LIN {X 0,Y 445.877,Z 691.903,A -85,B 0,C 180,E1 -8721.844,E2 -8721.844} C_VEL
LIN {X 0,Y 445.652,Z 697.529,A -85,B 0,C 180,E1 -8723.208,E2 -8723.208} C_VEL
LIN {X 0,Y 445.575,Z 701.931,A -85,B 0,C 180,E1 -8724.569,E2 -8724.569} C_VEL
LIN {X 0,Y 445.476,Z 704.248,A -85,B 0,C 180,E1 -8725.476,E2 -8725.476} C_VEL
LIN {X 0,Y 445.468,Z 706.135,A -85,B 0,C 180,E1 -8726.382,E2 -8726.382} C_VEL
LIN {X 0,Y 445.487,Z 707.56,A -85,B 0,C 180,E1 -8727.287,E2 -8727.287} C_VEL
LIN {X 0,Y 445.395,Z 709.177,A -85,B 0,C 180,E1 -8729.096,E2 -8729.096} C_VEL
LIN {X 0,Y 445.415,Z 709.398,A -85,B 0,C 180,E1 -8730,E2 -8730} C_VEL
LIN {X 0,Y 445.434,Z 709.177,A -85,B 0,C 180,E1 -8730.904,E2 -8730.904} C_VEL
LIN {X 0,Y 445.493,Z 707.56,A -85,B 0,C 180,E1 -8732.713,E2 -8732.713} C_VEL
LIN {X 0,Y 445.478,Z 706.134,A -85,B 0,C 180,E1 -8733.618,E2 -8733.618} C_VEL
LIN {X 0,Y 445.558,Z 703.166,A -85,B 0,C 180,E1 -8734.977,E2 -8734.977} C_VEL
LIN {X 0,Y 445.627,Z 698.572,A -85,B 0,C 180,E1 -8736.496,E2 -8736.496} C_VEL
LIN {X 0,Y 445.881,Z 691.901,A -85,B 0,C 180,E1 -8738.155,E2 -8738.155} C_VEL
LIN {X 0,Y 446.193,Z 684.816,A -85,B 0,C 180,E1 -8739.52,E2 -8739.52} C_VEL
LIN {X 0,Y 446.626,Z 675.955,A -85,B 0,C 180,E1 -8740.884,E2 -8740.884} C_VEL
LIN {X 0,Y 447.161,Z 666.837,A -85,B 0,C 180,E1 -8742.02,E2 -8742.02} C_VEL
LIN {X 0,Y 447.743,Z 655.911,A -85,B 0,C 180,E1 -8743.108,E2 -8743.108} C_VEL
LIN {X 0,Y 448.243,Z 645.348,A -85,B 0,C 180,E1 -8743.949,E2 -8743.949} C_VEL
LIN {X 0,Y 448.735,Z 633.519,A -85,B 0,C 180,E1 -8744.686,E2 -8744.686} C_VEL
LIN {X 0,Y 449.209,Z 620.349,A -85,B 0,C 180,E1 -8745.279,E2 -8745.279} C_VEL
LIN {X 0,Y 449.541,Z 608.315,A -85,B 0,C 180,E1 -8745.645,E2 -8745.645} C_VEL
LIN {X 0,Y 449.98,Z 567.208,A -85,B 0,C 180,E1 -8746.328,E2 -8746.328} C_VEL
LIN {X 0,Y 450.253,Z 534.372,A -85,B 0,C 180,E1 -8746.887,E2 -8746.887} C_VEL
LIN {X 0,Y 450.479,Z 513.135,A -85,B 0,C 180,E1 -8747.309,E2 -8747.309} C_VEL
LIN {X 0,Y 447.627,Z 483.502,A -85,B 0,C 180,E1 -8748.061,E2 -8748.061} C_VEL
LIN {X 0,Y 447.327,Z 480.598,A -85,B 0,C 180,E1 -8748.184,E2 -8748.184} C_VEL
LIN {X 0,Y 448.232,Z 456.008,A -85,B 0,C 180,E1 -8751.621,E2 -8751.621} C_VEL
LIN {X 0,Y 449.365,Z 434.276,A -85,B 0,C 180,E1 -8754.758,E2 -8754.758} C_VEL
LIN {X 0,Y 450.768,Z 413.421,A -85,B 0,C 180,E1 -8757.887,E2 -8757.887} C_VEL
LIN {X 0,Y 449.482,Z 405.511,A -85,B 0,C 180,E1 -8759.25,E2 -8759.25} C_VEL
LIN {X 0,Y 446.902,Z 394.819,A -85,B 0,C 180,E1 -8761.263,E2 -8761.263} C_VEL
LIN {X 0,Y 446.417,Z 392.958,A -85,B 0,C 180,E1 -8761.686,E2 -8761.686} C_VEL
LIN {X 0,Y 446.412,Z 392.881,A -85,B 0,C 180,E1 -8764.525,E2 -8764.525} C_VEL
LIN {X 0,Y 446.389,Z 392.884,A -85,B 0,C 180,E1 -8767.881,E2 -8767.881} C_VEL
LIN {X 0,Y 446.395,Z 392.878,A -85,B 0,C 180,E1 -8770.913,E2 -8770.913} C_VEL
LIN {X 0,Y 446.391,Z 392.882,A -85,B 0,C 180,E1 -8773.847,E2 -8773.847} C_VEL
LIN {X 0,Y 446.386,Z 392.879,A -85,B 0,C 180,E1 -8776.405,E2 -8776.405} C_VEL
LIN {X 0,Y 446.399,Z 392.88,A -85,B 0,C 180,E1 -8779.797,E2 -8779.797} C_VEL
LIN {X 0,Y 446.396,Z 392.882,A -85,B 0,C 180,E1 -8783.254,E2 -8783.254} C_VEL
LIN {X 0,Y 446.45,Z 392.872,A -85,B 0,C 180,E1 -8786.566,E2 -8786.566} C_VEL
LIN {X 0,Y 446.43,Z 392.877,A -85,B 0,C 180,E1 -8789.98,E2 -8789.98} C_VEL
LIN {X 0,Y 446.447,Z 392.873,A -85,B 0,C 180,E1 -8792.837,E2 -8792.837} C_VEL
LIN {X 0,Y 446.463,Z 392.873,A -85,B 0,C 180,E1 -8795.925,E2 -8795.925} C_VEL
LIN {X 0,Y 446.456,Z 392.874,A -85,B 0,C 180,E1 -8798.773,E2 -8798.773} C_VEL
LIN {X 0,Y 446.504,Z 392.971,A -85,B 0,C 180,E1 -8802.173,E2 -8802.173} C_VEL
LIN {X 0,Y 446.675,Z 393.84,A -85,B 0,C 180,E1 -8802.346,E2 -8802.346} C_VEL
LIN {X 0,Y 451.59,Z 405.892,A -85,B 0,C 180,E1 -8802.9,E2 -8802.9} C_VEL
LIN {X 0,Y 450.382,Z 476.779,A -85,B 0,C 180,E1 -8804.327,E2 -8804.327} C_VEL
LIN {X 0,Y 450.3,Z 489.562,A -85,B 0,C 180,E1 -8804.73,E2 -8804.73} C_VEL
LIN {X 0,Y 450.103,Z 503.008,A -85,B 0,C 180,E1 -8805.359,E2 -8805.359} C_VEL
LIN {X 0,Y 449.851,Z 513.751,A -85,B 0,C 180,E1 -8806.03,E2 -8806.03} C_VEL
LIN {X 0,Y 449.45,Z 524.679,A -85,B 0,C 180,E1 -8806.895,E2 -8806.895} C_VEL
LIN {X 0,Y 448.972,Z 533.964,A -85,B 0,C 180,E1 -8807.8,E2 -8807.8} C_VEL
LIN {X 0,Y 448.559,Z 543.404,A -85,B 0,C 180,E1 -8808.934,E2 -8808.934} C_VEL
LIN {X 0,Y 448.065,Z 551.12,A -85,B 0,C 180,E1 -8810.065,E2 -8810.065} C_VEL
LIN {X 0,Y 447.706,Z 558.821,A -85,B 0,C 180,E1 -8811.48,E2 -8811.48} C_VEL
LIN {X 0,Y 447.329,Z 564.472,A -85,B 0,C 180,E1 -8812.78,E2 -8812.78} C_VEL
LIN {X 0,Y 447.07,Z 569.094,A -85,B 0,C 180,E1 -8814.135,E2 -8814.135} C_VEL
LIN {X 0,Y 446.694,Z 572.607,A -85,B 0,C 180,E1 -8815.488,E2 -8815.488} C_VEL
LIN {X 0,Y 446.742,Z 574.35,A -85,B 0,C 180,E1 -8816.392,E2 -8816.392} C_VEL
LIN {X 0,Y 446.596,Z 575.652,A -85,B 0,C 180,E1 -8817.294,E2 -8817.294} C_VEL
LIN {X 0,Y 446.502,Z 576.521,A -85,B 0,C 180,E1 -8818.196,E2 -8818.196} C_VEL
LIN {X 0,Y 446.405,Z 576.994,A -85,B 0,C 180,E1 -8819.098,E2 -8819.098} C_VEL
LIN {X 0,Y 446.363,Z 577.045,A -85,B 0,C 180,E1 -8820,E2 -8820} C_VEL
LIN {X 0,Y 446.38,Z 576.645,A -85,B 0,C 180,E1 -8820.902,E2 -8820.902} C_VEL
LIN {X 0,Y 446.301,Z 575.861,A -85,B 0,C 180,E1 -8821.805,E2 -8821.805} C_VEL
LIN {X 0,Y 446.424,Z 574.653,A -85,B 0,C 180,E1 -8822.707,E2 -8822.707} C_VEL
LIN {X 0,Y 446.411,Z 572.035,A -85,B 0,C 180,E1 -8824.063,E2 -8824.063} C_VEL
LIN {X 0,Y 446.568,Z 568.375,A -85,B 0,C 180,E1 -8825.418,E2 -8825.418} C_VEL
LIN {X 0,Y 446.892,Z 562.968,A -85,B 0,C 180,E1 -8826.919,E2 -8826.919} C_VEL
LIN {X 0,Y 447.153,Z 556.334,A -85,B 0,C 180,E1 -8828.36,E2 -8828.36} C_VEL
LIN {X 0,Y 447.458,Z 548.495,A -85,B 0,C 180,E1 -8829.721,E2 -8829.721} C_VEL
LIN {X 0,Y 447.788,Z 540.446,A -85,B 0,C 180,E1 -8830.856,E2 -8830.856} C_VEL
LIN {X 0,Y 448.184,Z 530.608,A -85,B 0,C 180,E1 -8831.992,E2 -8831.992} C_VEL
LIN {X 0,Y 448.612,Z 519.67,A -85,B 0,C 180,E1 -8833.015,E2 -8833.015} C_VEL
LIN {X 0,Y 448.905,Z 508.7,A -85,B 0,C 180,E1 -8833.836,E2 -8833.836} C_VEL
LIN {X 0,Y 449.181,Z 496.311,A -85,B 0,C 180,E1 -8834.556,E2 -8834.556} C_VEL
LIN {X 0,Y 449.417,Z 483.722,A -85,B 0,C 180,E1 -8835.098,E2 -8835.098} C_VEL
LIN {X 0,Y 449.495,Z 470.727,A -85,B 0,C 180,E1 -8835.473,E2 -8835.473} C_VEL
LIN {X 0,Y 450.128,Z 404.106,A -85,B 0,C 180,E1 -8836.708,E2 -8836.708} C_VEL
LIN {X 0,Y 446.657,Z 393.7,A -85,B 0,C 180,E1 -8837.05,E2 -8837.05} C_VEL
LIN {X 0,Y 446.482,Z 392.961,A -85,B 0,C 180,E1 -8837.209,E2 -8837.209} C_VEL
LIN {X 0,Y 446.447,Z 392.875,A -85,B 0,C 180,E1 -8840.263,E2 -8840.263} C_VEL
LIN {X 0,Y 446.431,Z 392.876,A -85,B 0,C 180,E1 -8843.177,E2 -8843.177} C_VEL
LIN {X 0,Y 446.441,Z 392.873,A -85,B 0,C 180,E1 -8846.193,E2 -8846.193} C_VEL
LIN {X 0,Y 446.44,Z 392.868,A -85,B 0,C 180,E1 -8849.21,E2 -8849.21} C_VEL
LIN {X 0,Y 446.422,Z 392.877,A -85,B 0,C 180,E1 -8852.362,E2 -8852.362} C_VEL
LIN {X 0,Y 446.42,Z 392.874,A -85,B 0,C 180,E1 -8855.626,E2 -8855.626} C_VEL
LIN {X 0,Y 446.443,Z 392.874,A -85,B 0,C 180,E1 -8859.027,E2 -8859.027} C_VEL
LIN {X 0,Y 446.423,Z 392.872,A -85,B 0,C 180,E1 -8862.275,E2 -8862.275} C_VEL
LIN {X 0,Y 446.452,Z 392.869,A -85,B 0,C 180,E1 -8865.104,E2 -8865.104} C_VEL
LIN {X 0,Y 446.421,Z 392.877,A -85,B 0,C 180,E1 -8868.608,E2 -8868.608} C_VEL
LIN {X 0,Y 446.413,Z 392.865,A -85,B 0,C 180,E1 -8871.922,E2 -8871.922} C_VEL
LIN {X 0,Y 446.431,Z 392.869,A -85,B 0,C 180,E1 -8875.477,E2 -8875.477} C_VEL
LIN {X 0,Y 446.488,Z 392.994,A -85,B 0,C 180,E1 -8879.117,E2 -8879.117} C_VEL
LIN {X 0,Y 449.858,Z 407.067,A -85,B 0,C 180,E1 -8881.314,E2 -8881.314} C_VEL
LIN {X 0,Y 451.299,Z 414.583,A -85,B 0,C 180,E1 -8882.448,E2 -8882.448} C_VEL
LIN {X 0,Y 450.315,Z 437.381,A -85,B 0,C 180,E1 -8885.57,E2 -8885.57} C_VEL
LIN {X 0,Y 449.475,Z 456.758,A -85,B 0,C 180,E1 -8888.201,E2 -8888.201} C_VEL
LIN {X 0,Y 448.796,Z 474.172,A -85,B 0,C 180,E1 -8890.501,E2 -8890.501} C_VEL
LIN {X 0,Y 448.016,Z 477.382,A -85,B 0,C 180,E1 -8890.88,E2 -8890.88} C_VEL
LIN {X 0,Y 444.945,Z 482.695,A -85,B 0,C 180,E1 -8891.434,E2 -8891.434} C_VEL
LIN {X 0,Y 442.344,Z 487.283,A -85,B 0,C 180,E1 -8891.854,E2 -8891.854} C_VEL
LIN {X 0,Y 441.926,Z 490.019,A -85,B 0,C 180,E1 -8891.993,E2 -8891.993} C_VEL
LIN {X 0,Y 441.979,Z 490.598,A -85,B 0,C 180,E1 -8892.008,E2 -8892.008} C_VEL
LIN {X 0,Y 444.18,Z 506.961,A -85,B 0,C 180,E1 -8892.374,E2 -8892.374} C_VEL
LIN {X 0,Y 443.246,Z 598.809,A -85,B 0,C 180,E1 -8893.89,E2 -8893.89} C_VEL
LIN {X 0,Y 442.885,Z 612.281,A -85,B 0,C 180,E1 -8894.291,E2 -8894.291} C_VEL
LIN {X 0,Y 442.359,Z 624.85,A -85,B 0,C 180,E1 -8894.862,E2 -8894.862} C_VEL
LIN {X 0,Y 441.775,Z 636.976,A -85,B 0,C 180,E1 -8895.607,E2 -8895.607} C_VEL
LIN {X 0,Y 441.233,Z 648.191,A -85,B 0,C 180,E1 -8896.504,E2 -8896.504} C_VEL
LIN {X 0,Y 440.634,Z 658.741,A -85,B 0,C 180,E1 -8897.566,E2 -8897.566} C_VEL
LIN {X 0,Y 439.971,Z 668.052,A -85,B 0,C 180,E1 -8898.716,E2 -8898.716} C_VEL
LIN {X 0,Y 439.426,Z 677.035,A -85,B 0,C 180,E1 -8900.1,E2 -8900.1} C_VEL
LIN {X 0,Y 438.986,Z 684.246,A -85,B 0,C 180,E1 -8901.484,E2 -8901.484} C_VEL
LIN {X 0,Y 438.719,Z 689.142,A -85,B 0,C 180,E1 -8902.637,E2 -8902.637} C_VEL
LIN {X 0,Y 438.555,Z 693.879,A -85,B 0,C 180,E1 -8904.021,E2 -8904.021} C_VEL
LIN {X 0,Y 438.375,Z 697.508,A -85,B 0,C 180,E1 -8905.402,E2 -8905.402} C_VEL
LIN {X 0,Y 438.307,Z 699.376,A -85,B 0,C 180,E1 -8906.323,E2 -8906.323} C_VEL
LIN {X 0,Y 438.346,Z 700.805,A -85,B 0,C 180,E1 -8907.243,E2 -8907.243} C_VEL
LIN {X 0,Y 438.231,Z 702.424,A -85,B 0,C 180,E1 -8909.081,E2 -8909.081} C_VEL
LIN {X 0,Y 438.229,Z 702.662,A -85,B 0,C 180,E1 -8910,E2 -8910} C_VEL
LIN {X 0,Y 438.231,Z 702.471,A -85,B 0,C 180,E1 -8910.919,E2 -8910.919} C_VEL
LIN {X 0,Y 438.346,Z 700.914,A -85,B 0,C 180,E1 -8912.757,E2 -8912.757} C_VEL
LIN {X 0,Y 438.307,Z 699.546,A -85,B 0,C 180,E1 -8913.677,E2 -8913.677} C_VEL
LIN {X 0,Y 438.448,Z 696.666,A -85,B 0,C 180,E1 -8915.058,E2 -8915.058} C_VEL
LIN {X 0,Y 438.547,Z 692.602,A -85,B 0,C 180,E1 -8916.488,E2 -8916.488} C_VEL
LIN {X 0,Y 438.766,Z 687.691,A -85,B 0,C 180,E1 -8917.825,E2 -8917.825} C_VEL
LIN {X 0,Y 439.161,Z 681.306,A -85,B 0,C 180,E1 -8919.209,E2 -8919.209} C_VEL
LIN {X 0,Y 439.625,Z 673.378,A -85,B 0,C 180,E1 -8920.594,E2 -8920.594} C_VEL
LIN {X 0,Y 440.164,Z 665.28,A -85,B 0,C 180,E1 -8921.746,E2 -8921.746} C_VEL
LIN {X 0,Y 440.869,Z 655.338,A -85,B 0,C 180,E1 -8922.896,E2 -8922.896} C_VEL
LIN {X 0,Y 441.388,Z 644.17,A -85,B 0,C 180,E1 -8923.936,E2 -8923.936} C_VEL
LIN {X 0,Y 441.985,Z 633.248,A -85,B 0,C 180,E1 -8924.739,E2 -8924.739} C_VEL
LIN {X 0,Y 442.566,Z 620.993,A -85,B 0,C 180,E1 -8925.426,E2 -8925.426} C_VEL
LIN {X 0,Y 443.06,Z 608.283,A -85,B 0,C 180,E1 -8925.939,E2 -8925.939} C_VEL
LIN {X 0,Y 443.367,Z 594.914,A -85,B 0,C 180,E1 -8926.283,E2 -8926.283} C_VEL
LIN {X 0,Y 444.09,Z 505.201,A -85,B 0,C 180,E1 -8927.753,E2 -8927.753} C_VEL
LIN {X 0,Y 441.619,Z 487.767,A -85,B 0,C 180,E1 -8928.168,E2 -8928.168} C_VEL
LIN {X 0,Y 442.206,Z 467.995,A -85,B 0,C 180,E1 -8930.709,E2 -8930.709} C_VEL
LIN {X 0,Y 443.215,Z 444.829,A -85,B 0,C 180,E1 -8933.851,E2 -8933.851} C_VEL
LIN {X 0,Y 444.211,Z 423.493,A -85,B 0,C 180,E1 -8936.802,E2 -8936.802} C_VEL
LIN {X 0,Y 444.469,Z 415.37,A -85,B 0,C 180,E1 -8937.929,E2 -8937.929} C_VEL
LIN {X 0,Y 441.016,Z 400.06,A -85,B 0,C 180,E1 -8940.285,E2 -8940.285} C_VEL
LIN {X 0,Y 439.416,Z 393.899,A -85,B 0,C 180,E1 -8941.286,E2 -8941.286} C_VEL
LIN {X 0,Y 439.387,Z 393.749,A -85,B 0,C 180,E1 -8944.044,E2 -8944.044} C_VEL
LIN {X 0,Y 439.341,Z 393.751,A -85,B 0,C 180,E1 -8946.885,E2 -8946.885} C_VEL
LIN {X 0,Y 439.348,Z 393.748,A -85,B 0,C 180,E1 -8949.84,E2 -8949.84} C_VEL
LIN {X 0,Y 439.335,Z 393.758,A -85,B 0,C 180,E1 -8952.62,E2 -8952.62} C_VEL
LIN {X 0,Y 439.379,Z 393.738,A -85,B 0,C 180,E1 -8955.268,E2 -8955.268} C_VEL
LIN {X 0,Y 439.369,Z 393.753,A -85,B 0,C 180,E1 -8958.747,E2 -8958.747} C_VEL
LIN {X 0,Y 439.362,Z 393.757,A -85,B 0,C 180,E1 -8961.611,E2 -8961.611} C_VEL
LIN {X 0,Y 439.397,Z 393.749,A -85,B 0,C 180,E1 -8964.844,E2 -8964.844} C_VEL
LIN {X 0,Y 439.373,Z 393.755,A -85,B 0,C 180,E1 -8968.139,E2 -8968.139} C_VEL
LIN {X 0,Y 439.385,Z 393.746,A -85,B 0,C 180,E1 -8971.324,E2 -8971.324} C_VEL
LIN {X 0,Y 439.374,Z 393.752,A -85,B 0,C 180,E1 -8974.413,E2 -8974.413} C_VEL
LIN {X 0,Y 439.367,Z 393.748,A -85,B 0,C 180,E1 -8977.425,E2 -8977.425} C_VEL
LIN {X 0,Y 439.445,Z 393.74,A -85,B 0,C 180,E1 -8980.663,E2 -8980.663} C_VEL
LIN {X 0,Y 439.424,Z 393.747,A -85,B 0,C 180,E1 -8984.223,E2 -8984.223} C_VEL
LIN {X 0,Y 439.488,Z 393.737,A -85,B 0,C 180,E1 -8987.286,E2 -8987.286} C_VEL
LIN {X 0,Y 439.479,Z 393.736,A -85,B 0,C 180,E1 -8990.798,E2 -8990.798} C_VEL
LIN {X 0,Y 439.562,Z 393.729,A -85,B 0,C 180,E1 -8993.574,E2 -8993.574} C_VEL
LIN {X 0,Y 439.406,Z 393.737,A -85,B 0,C 180,E1 -8995.413,E2 -8995.413} C_VEL
LIN {X 0,Y 439.629,Z 393.722,A -85,B 0,C 180,E1 -8998.168,E2 -8998.168} C_VEL
LIN {X 0,Y 439.672,Z 393.714,A -85,B 0,C 180,E1 -9000,E2 -9000} C_VEL
LIN {X 0,Y 439.607,Z 393.708,A -85,B 0,C 180,E1 -9002.749,E2 -9002.749} C_VEL
LIN {X 0,Y 439.562,Z 393.728,A -85,B 0,C 180,E1 -9006.426,E2 -9006.426} C_VEL
LIN {X 0,Y 439.478,Z 393.731,A -85,B 0,C 180,E1 -9009.202,E2 -9009.202} C_VEL
LIN {X 0,Y 439.467,Z 393.739,A -85,B 0,C 180,E1 -9012.938,E2 -9012.938} C_VEL
LIN {X 0,Y 439.399,Z 393.736,A -85,B 0,C 180,E1 -9016.325,E2 -9016.325} C_VEL
LIN {X 0,Y 439.372,Z 393.755,A -85,B 0,C 180,E1 -9019.628,E2 -9019.628} C_VEL
LIN {X 0,Y 439.362,Z 393.742,A -85,B 0,C 180,E1 -9022.576,E2 -9022.576} C_VEL
LIN {X 0,Y 439.357,Z 393.756,A -85,B 0,C 180,E1 -9025.588,E2 -9025.588} C_VEL
LIN {X 0,Y 439.384,Z 393.74,A -85,B 0,C 180,E1 -9028.676,E2 -9028.676} C_VEL
LIN {X 0,Y 439.368,Z 393.756,A -85,B 0,C 180,E1 -9032.029,E2 -9032.029} C_VEL
LIN {X 0,Y 439.389,Z 393.745,A -85,B 0,C 180,E1 -9035.338,E2 -9035.338} C_VEL
LIN {X 0,Y 439.35,Z 393.749,A -85,B 0,C 180,E1 -9038.599,E2 -9038.599} C_VEL
LIN {X 0,Y 439.346,Z 393.732,A -85,B 0,C 180,E1 -9042.21,E2 -9042.21} C_VEL
LIN {X 0,Y 439.373,Z 393.753,A -85,B 0,C 180,E1 -9045.267,E2 -9045.267} C_VEL
LIN {X 0,Y 439.359,Z 393.729,A -85,B 0,C 180,E1 -9048.748,E2 -9048.748} C_VEL
LIN {X 0,Y 439.353,Z 393.756,A -85,B 0,C 180,E1 -9051.612,E2 -9051.612} C_VEL
LIN {X 0,Y 439.388,Z 393.753,A -85,B 0,C 180,E1 -9054.843,E2 -9054.843} C_VEL
LIN {X 0,Y 439.389,Z 393.934,A -85,B 0,C 180,E1 -9058.359,E2 -9058.359} C_VEL
LIN {X 0,Y 443.711,Z 412.535,A -85,B 0,C 180,E1 -9061.407,E2 -9061.407} C_VEL
LIN {X 0,Y 444.061,Z 417.576,A -85,B 0,C 180,E1 -9062.171,E2 -9062.171} C_VEL
LIN {X 0,Y 442.664,Z 439.939,A -85,B 0,C 180,E1 -9065.383,E2 -9065.383} C_VEL
LIN {X 0,Y 441.484,Z 462.058,A -85,B 0,C 180,E1 -9068.522,E2 -9068.522} C_VEL
LIN {X 0,Y 440.487,Z 486.126,A -85,B 0,C 180,E1 -9071.888,E2 -9071.888} C_VEL
LIN {X 0,Y 440.734,Z 489.285,A -85,B 0,C 180,E1 -9072.018,E2 -9072.018} C_VEL
LIN {X 0,Y 443.561,Z 515.823,A -85,B 0,C 180,E1 -9072.577,E2 -9072.577} C_VEL
LIN {X 0,Y 442.755,Z 607.315,A -85,B 0,C 180,E1 -9074.079,E2 -9074.079} C_VEL
LIN {X 0,Y 442.367,Z 620.411,A -85,B 0,C 180,E1 -9074.478,E2 -9074.478} C_VEL
LIN {X 0,Y 441.883,Z 633.544,A -85,B 0,C 180,E1 -9075.081,E2 -9075.081} C_VEL
LIN {X 0,Y 441.325,Z 645.346,A -85,B 0,C 180,E1 -9075.827,E2 -9075.827} C_VEL
LIN {X 0,Y 440.771,Z 656.588,A -85,B 0,C 180,E1 -9076.743,E2 -9076.743} C_VEL
LIN {X 0,Y 440.167,Z 666.82,A -85,B 0,C 180,E1 -9077.786,E2 -9077.786} C_VEL
LIN {X 0,Y 439.64,Z 675.926,A -85,B 0,C 180,E1 -9078.94,E2 -9078.94} C_VEL
LIN {X 0,Y 439.166,Z 684.77,A -85,B 0,C 180,E1 -9080.326,E2 -9080.326} C_VEL
LIN {X 0,Y 438.841,Z 691.853,A -85,B 0,C 180,E1 -9081.713,E2 -9081.713} C_VEL
LIN {X 0,Y 438.588,Z 697.476,A -85,B 0,C 180,E1 -9083.097,E2 -9083.097} C_VEL
LIN {X 0,Y 438.49,Z 701.879,A -85,B 0,C 180,E1 -9084.481,E2 -9084.481} C_VEL
LIN {X 0,Y 438.403,Z 704.195,A -85,B 0,C 180,E1 -9085.402,E2 -9085.402} C_VEL
LIN {X 0,Y 438.366,Z 706.082,A -85,B 0,C 180,E1 -9086.323,E2 -9086.323} C_VEL
LIN {X 0,Y 438.412,Z 707.507,A -85,B 0,C 180,E1 -9087.243,E2 -9087.243} C_VEL
LIN {X 0,Y 438.306,Z 709.124,A -85,B 0,C 180,E1 -9089.081,E2 -9089.081} C_VEL
LIN {X 0,Y 438.322,Z 709.343,A -85,B 0,C 180,E1 -9090,E2 -9090} C_VEL
LIN {X 0,Y 438.342,Z 709.123,A -85,B 0,C 180,E1 -9090.919,E2 -9090.919} C_VEL
LIN {X 0,Y 438.419,Z 707.506,A -85,B 0,C 180,E1 -9092.756,E2 -9092.756} C_VEL
LIN {X 0,Y 438.377,Z 706.08,A -85,B 0,C 180,E1 -9093.677,E2 -9093.677} C_VEL
LIN {X 0,Y 438.489,Z 703.113,A -85,B 0,C 180,E1 -9095.057,E2 -9095.057} C_VEL
LIN {X 0,Y 438.546,Z 698.917,A -85,B 0,C 180,E1 -9096.488,E2 -9096.488} C_VEL
LIN {X 0,Y 438.767,Z 692.855,A -85,B 0,C 180,E1 -9098.057,E2 -9098.057} C_VEL
LIN {X 0,Y 439.092,Z 686.058,A -85,B 0,C 180,E1 -9099.442,E2 -9099.442} C_VEL
LIN {X 0,Y 439.466,Z 679.096,A -85,B 0,C 180,E1 -9100.598,E2 -9100.598} C_VEL
LIN {X 0,Y 439.966,Z 670.675,A -85,B 0,C 180,E1 -9101.751,E2 -9101.751} C_VEL
LIN {X 0,Y 440.573,Z 660.238,A -85,B 0,C 180,E1 -9102.904,E2 -9102.904} C_VEL
LIN {X 0,Y 441.108,Z 649.882,A -85,B 0,C 180,E1 -9103.827,E2 -9103.827} C_VEL
LIN {X 0,Y 441.64,Z 638.443,A -85,B 0,C 180,E1 -9104.633,E2 -9104.633} C_VEL
LIN {X 0,Y 442.183,Z 626.534,A -85,B 0,C 180,E1 -9105.262,E2 -9105.262} C_VEL
LIN {X 0,Y 442.575,Z 613.624,A -85,B 0,C 180,E1 -9105.75,E2 -9105.75} C_VEL
LIN {X 0,Y 442.828,Z 601.37,A -85,B 0,C 180,E1 -9106.036,E2 -9106.036} C_VEL
LIN {X 0,Y 443.401,Z 541.215,A -85,B 0,C 180,E1 -9107.037,E2 -9107.037} C_VEL
LIN {X 0,Y 443.774,Z 513.924,A -85,B 0,C 180,E1 -9107.592,E2 -9107.592} C_VEL
LIN {X 0,Y 441.024,Z 484.788,A -85,B 0,C 180,E1 -9108.362,E2 -9108.362} C_VEL
LIN {X 0,Y 440.345,Z 479.393,A -85,B 0,C 180,E1 -9108.548,E2 -9108.548} C_VEL
LIN {X 0,Y 441.272,Z 457.008,A -85,B 0,C 180,E1 -9111.734,E2 -9111.734} C_VEL
LIN {X 0,Y 442.519,Z 434.905,A -85,B 0,C 180,E1 -9115,E2 -9115} C_VEL
LIN {X 0,Y 443.968,Z 414.817,A -85,B 0,C 180,E1 -9118.095,E2 -9118.095} C_VEL
LIN {X 0,Y 442.313,Z 405.461,A -85,B 0,C 180,E1 -9119.771,E2 -9119.771} C_VEL
LIN {X 0,Y 439.632,Z 395.042,A -85,B 0,C 180,E1 -9121.84,E2 -9121.84} C_VEL
LIN {X 0,Y 439.377,Z 393.861,A -85,B 0,C 180,E1 -9122.122,E2 -9122.122} C_VEL
LIN {X 0,Y 439.383,Z 393.755,A -85,B 0,C 180,E1 -9125.338,E2 -9125.338} C_VEL
LIN {X 0,Y 439.35,Z 393.759,A -85,B 0,C 180,E1 -9128.599,E2 -9128.599} C_VEL
LIN {X 0,Y 439.358,Z 393.757,A -85,B 0,C 180,E1 -9131.252,E2 -9131.252} C_VEL
LIN {X 0,Y 439.376,Z 393.753,A -85,B 0,C 180,E1 -9134.733,E2 -9134.733} C_VEL
LIN {X 0,Y 439.349,Z 393.76,A -85,B 0,C 180,E1 -9137.79,E2 -9137.79} C_VEL
LIN {X 0,Y 439.359,Z 393.759,A -85,B 0,C 180,E1 -9141.402,E2 -9141.402} C_VEL
LIN {X 0,Y 439.396,Z 393.752,A -85,B 0,C 180,E1 -9144.844,E2 -9144.844} C_VEL
LIN {X 0,Y 439.374,Z 393.755,A -85,B 0,C 180,E1 -9148.14,E2 -9148.14} C_VEL
LIN {X 0,Y 439.411,Z 393.752,A -85,B 0,C 180,E1 -9151.604,E2 -9151.604} C_VEL
LIN {X 0,Y 439.379,Z 393.752,A -85,B 0,C 180,E1 -9154.413,E2 -9154.413} C_VEL
LIN {X 0,Y 439.366,Z 393.758,A -85,B 0,C 180,E1 -9157.425,E2 -9157.425} C_VEL
LIN {X 0,Y 439.443,Z 393.749,A -85,B 0,C 180,E1 -9160.663,E2 -9160.663} C_VEL
LIN {X 0,Y 439.469,Z 393.977,A -85,B 0,C 180,E1 -9161.83,E2 -9161.83} C_VEL
LIN {X 0,Y 439.709,Z 394.984,A -85,B 0,C 180,E1 -9161.975,E2 -9161.975} C_VEL
LIN {X 0,Y 444.96,Z 407.288,A -85,B 0,C 180,E1 -9162.572,E2 -9162.572} C_VEL
LIN {X 0,Y 443.725,Z 478.354,A -85,B 0,C 180,E1 -9164.056,E2 -9164.056} C_VEL
LIN {X 0,Y 443.645,Z 491.663,A -85,B 0,C 180,E1 -9164.495,E2 -9164.495} C_VEL
LIN {X 0,Y 443.401,Z 504.246,A -85,B 0,C 180,E1 -9165.098,E2 -9165.098} C_VEL
LIN {X 0,Y 443.137,Z 515.067,A -85,B 0,C 180,E1 -9165.787,E2 -9165.787} C_VEL
LIN {X 0,Y 442.673,Z 526.201,A -85,B 0,C 180,E1 -9166.691,E2 -9166.691} C_VEL
LIN {X 0,Y 442.126,Z 536.421,A -85,B 0,C 180,E1 -9167.725,E2 -9167.725} C_VEL
LIN {X 0,Y 441.718,Z 544.745,A -85,B 0,C 180,E1 -9168.761,E2 -9168.761} C_VEL
LIN {X 0,Y 441.213,Z 552.431,A -85,B 0,C 180,E1 -9169.909,E2 -9169.909} C_VEL
LIN {X 0,Y 440.823,Z 559.831,A -85,B 0,C 180,E1 -9171.289,E2 -9171.289} C_VEL
LIN {X 0,Y 440.397,Z 565.725,A -85,B 0,C 180,E1 -9172.665,E2 -9172.665} C_VEL
LIN {X 0,Y 440.114,Z 570.319,A -85,B 0,C 180,E1 -9174.042,E2 -9174.042} C_VEL
LIN {X 0,Y 439.742,Z 573.795,A -85,B 0,C 180,E1 -9175.417,E2 -9175.417} C_VEL
LIN {X 0,Y 439.754,Z 575.51,A -85,B 0,C 180,E1 -9176.335,E2 -9176.335} C_VEL
LIN {X 0,Y 439.599,Z 576.774,A -85,B 0,C 180,E1 -9177.251,E2 -9177.251} C_VEL
LIN {X 0,Y 439.491,Z 577.619,A -85,B 0,C 180,E1 -9178.167,E2 -9178.167} C_VEL
LIN {X 0,Y 439.388,Z 578.067,A -85,B 0,C 180,E1 -9179.084,E2 -9179.084} C_VEL
LIN {X 0,Y 439.34,Z 578.078,A -85,B 0,C 180,E1 -9180,E2 -9180} C_VEL
LIN {X 0,Y 439.357,Z 577.647,A -85,B 0,C 180,E1 -9180.917,E2 -9180.917} C_VEL
LIN {X 0,Y 439.278,Z 576.837,A -85,B 0,C 180,E1 -9181.834,E2 -9181.834} C_VEL
LIN {X 0,Y 439.403,Z 575.598,A -85,B 0,C 180,E1 -9182.75,E2 -9182.75} C_VEL
LIN {X 0,Y 439.386,Z 572.928,A -85,B 0,C 180,E1 -9184.128,E2 -9184.128} C_VEL
LIN {X 0,Y 439.566,Z 569.203,A -85,B 0,C 180,E1 -9185.505,E2 -9185.505} C_VEL
LIN {X 0,Y 439.879,Z 564.018,A -85,B 0,C 180,E1 -9186.956,E2 -9186.956} C_VEL
LIN {X 0,Y 440.158,Z 556.993,A -85,B 0,C 180,E1 -9188.493,E2 -9188.493} C_VEL
LIN {X 0,Y 440.492,Z 549.045,A -85,B 0,C 180,E1 -9189.876,E2 -9189.876} C_VEL
LIN {X 0,Y 440.812,Z 540.884,A -85,B 0,C 180,E1 -9191.03,E2 -9191.03} C_VEL
LIN {X 0,Y 441.238,Z 530.912,A -85,B 0,C 180,E1 -9192.184,E2 -9192.184} C_VEL
LIN {X 0,Y 441.705,Z 519.803,A -85,B 0,C 180,E1 -9193.222,E2 -9193.222} C_VEL
LIN {X 0,Y 441.98,Z 508.286,A -85,B 0,C 180,E1 -9194.076,E2 -9194.076} C_VEL
LIN {X 0,Y 442.295,Z 495.903,A -85,B 0,C 180,E1 -9194.787,E2 -9194.787} C_VEL
LIN {X 0,Y 442.523,Z 483.539,A -85,B 0,C 180,E1 -9195.31,E2 -9195.31} C_VEL
LIN {X 0,Y 442.579,Z 469.839,A -85,B 0,C 180,E1 -9195.691,E2 -9195.691} C_VEL
LIN {X 0,Y 443.25,Z 405.569,A -85,B 0,C 180,E1 -9196.905,E2 -9196.905} C_VEL
LIN {X 0,Y 439.58,Z 394.58,A -85,B 0,C 180,E1 -9197.278,E2 -9197.278} C_VEL
LIN {X 0,Y 439.43,Z 393.824,A -85,B 0,C 180,E1 -9197.451,E2 -9197.451} C_VEL
LIN {X 0,Y 439.392,Z 393.755,A -85,B 0,C 180,E1 -9200.603,E2 -9200.603} C_VEL
LIN {X 0,Y 439.415,Z 393.749,A -85,B 0,C 180,E1 -9204.264,E2 -9204.264} C_VEL
LIN {X 0,Y 439.388,Z 393.745,A -85,B 0,C 180,E1 -9207.636,E2 -9207.636} C_VEL
LIN {X 0,Y 439.363,Z 393.757,A -85,B 0,C 180,E1 -9210.789,E2 -9210.789} C_VEL
LIN {X 0,Y 439.387,Z 393.742,A -85,B 0,C 180,E1 -9214.044,E2 -9214.044} C_VEL
LIN {X 0,Y 439.35,Z 393.756,A -85,B 0,C 180,E1 -9216.887,E2 -9216.887} C_VEL
LIN {X 0,Y 439.404,Z 393.749,A -85,B 0,C 180,E1 -9219.849,E2 -9219.849} C_VEL
LIN {X 0,Y 439.372,Z 393.753,A -85,B 0,C 180,E1 -9222.625,E2 -9222.625} C_VEL
LIN {X 0,Y 439.4,Z 393.747,A -85,B 0,C 180,E1 -9225.27,E2 -9225.27} C_VEL
LIN {X 0,Y 439.383,Z 393.755,A -85,B 0,C 180,E1 -9228.744,E2 -9228.744} C_VEL
LIN {X 0,Y 439.366,Z 393.741,A -85,B 0,C 180,E1 -9231.609,E2 -9231.609} C_VEL
LIN {X 0,Y 439.4,Z 393.742,A -85,B 0,C 180,E1 -9234.844,E2 -9234.844} C_VEL
LIN {X 0,Y 439.375,Z 393.749,A -85,B 0,C 180,E1 -9238.14,E2 -9238.14} C_VEL
LIN {X 0,Y 439.446,Z 394.03,A -85,B 0,C 180,E1 -9238.851,E2 -9238.851} C_VEL
LIN {X 0,Y 443.13,Z 409.12,A -85,B 0,C 180,E1 -9241.213,E2 -9241.213} C_VEL
LIN {X 0,Y 444.511,Z 416.276,A -85,B 0,C 180,E1 -9242.301,E2 -9242.301} C_VEL
LIN {X 0,Y 443.453,Z 438.795,A -85,B 0,C 180,E1 -9245.416,E2 -9245.416} C_VEL
LIN {X 0,Y 442.508,Z 460.075,A -85,B 0,C 180,E1 -9248.33,E2 -9248.33} C_VEL
LIN {X 0,Y 441.634,Z 485.493,A -85,B 0,C 180,E1 -9251.658,E2 -9251.658} C_VEL
LIN {X 0,Y 441.643,Z 488.223,A -85,B 0,C 180,E1 -9251.948,E2 -9251.948} C_VEL
LIN {X 0,Y 441.979,Z 490.598,A -85,B 0,C 180,E1 -9252.008,E2 -9252.008} C_VEL
LIN {X 0,Y 442.085,Z 496.455,A -85,B 0,C 180,E1 -9252.111,E2 -9252.111} C_VEL
LIN {X 0,Y 440.226,Z 506.193,A -85,B 0,C 180,E1 -9252.198,E2 -9252.198} C_VEL
LIN {X 0,Y 437.57,Z 517.947,A -85,B 0,C 180,E1 -9252.286,E2 -9252.286} C_VEL
LIN {X 0,Y 437.257,Z 521.92,A -85,B 0,C 180,E1 -9252.34,E2 -9252.34} C_VEL
LIN {X 0,Y 436.45,Z 598.794,A -85,B 0,C 180,E1 -9253.633,E2 -9253.633} C_VEL
LIN {X 0,Y 436.044,Z 612.3,A -85,B 0,C 180,E1 -9254.038,E2 -9254.038} C_VEL
LIN {X 0,Y 435.511,Z 624.883,A -85,B 0,C 180,E1 -9254.618,E2 -9254.618} C_VEL
LIN {X 0,Y 434.9,Z 637.017,A -85,B 0,C 180,E1 -9255.374,E2 -9255.374} C_VEL
LIN {X 0,Y 434.296,Z 648.237,A -85,B 0,C 180,E1 -9256.284,E2 -9256.284} C_VEL
LIN {X 0,Y 433.681,Z 658.789,A -85,B 0,C 180,E1 -9257.363,E2 -9257.363} C_VEL
LIN {X 0,Y 433.005,Z 668.103,A -85,B 0,C 180,E1 -9258.532,E2 -9258.532} C_VEL
LIN {X 0,Y 432.407,Z 677.087,A -85,B 0,C 180,E1 -9259.938,E2 -9259.938} C_VEL
LIN {X 0,Y 431.962,Z 684.299,A -85,B 0,C 180,E1 -9261.344,E2 -9261.344} C_VEL
LIN {X 0,Y 431.613,Z 690.921,A -85,B 0,C 180,E1 -9262.985,E2 -9262.985} C_VEL
LIN {X 0,Y 431.443,Z 695.271,A -85,B 0,C 180,E1 -9264.391,E2 -9264.391} C_VEL
LIN {X 0,Y 431.308,Z 697.562,A -85,B 0,C 180,E1 -9265.327,E2 -9265.327} C_VEL
LIN {X 0,Y 431.213,Z 699.43,A -85,B 0,C 180,E1 -9266.262,E2 -9266.262} C_VEL
LIN {X 0,Y 431.243,Z 700.859,A -85,B 0,C 180,E1 -9267.198,E2 -9267.198} C_VEL
LIN {X 0,Y 431.203,Z 701.86,A -85,B 0,C 180,E1 -9268.132,E2 -9268.132} C_VEL
LIN {X 0,Y 431.144,Z 702.716,A -85,B 0,C 180,E1 -9270,E2 -9270} C_VEL
LIN {X 0,Y 431.149,Z 702.525,A -85,B 0,C 180,E1 -9270.934,E2 -9270.934} C_VEL
LIN {X 0,Y 431.204,Z 701.937,A -85,B 0,C 180,E1 -9271.868,E2 -9271.868} C_VEL
LIN {X 0,Y 431.243,Z 700.967,A -85,B 0,C 180,E1 -9272.803,E2 -9272.803} C_VEL
LIN {X 0,Y 431.213,Z 699.599,A -85,B 0,C 180,E1 -9273.738,E2 -9273.738} C_VEL
LIN {X 0,Y 431.385,Z 696.718,A -85,B 0,C 180,E1 -9275.141,E2 -9275.141} C_VEL
LIN {X 0,Y 431.483,Z 692.807,A -85,B 0,C 180,E1 -9276.547,E2 -9276.547} C_VEL
LIN {X 0,Y 431.729,Z 687.741,A -85,B 0,C 180,E1 -9277.954,E2 -9277.954} C_VEL
LIN {X 0,Y 432.121,Z 681.354,A -85,B 0,C 180,E1 -9279.36,E2 -9279.36} C_VEL
LIN {X 0,Y 432.627,Z 673.423,A -85,B 0,C 180,E1 -9280.767,E2 -9280.767} C_VEL
LIN {X 0,Y 433.207,Z 665.323,A -85,B 0,C 180,E1 -9281.938,E2 -9281.938} C_VEL
LIN {X 0,Y 433.947,Z 655.377,A -85,B 0,C 180,E1 -9283.105,E2 -9283.105} C_VEL
LIN {X 0,Y 434.49,Z 644.203,A -85,B 0,C 180,E1 -9284.161,E2 -9284.161} C_VEL
LIN {X 0,Y 435.135,Z 633.273,A -85,B 0,C 180,E1 -9284.977,E2 -9284.977} C_VEL
LIN {X 0,Y 435.736,Z 621.003,A -85,B 0,C 180,E1 -9285.674,E2 -9285.674} C_VEL
LIN {X 0,Y 436.26,Z 608.271,A -85,B 0,C 180,E1 -9286.195,E2 -9286.195} C_VEL
LIN {X 0,Y 436.537,Z 596.365,A -85,B 0,C 180,E1 -9286.515,E2 -9286.515} C_VEL
LIN {X 0,Y 437.359,Z 506.215,A -85,B 0,C 180,E1 -9288.016,E2 -9288.016} C_VEL
LIN {X 0,Y 434.716,Z 487.651,A -85,B 0,C 180,E1 -9288.475,E2 -9288.475} C_VEL
LIN {X 0,Y 435.379,Z 467.839,A -85,B 0,C 180,E1 -9291.049,E2 -9291.049} C_VEL
LIN {X 0,Y 436.432,Z 444.512,A -85,B 0,C 180,E1 -9294.245,E2 -9294.245} C_VEL
LIN {X 0,Y 437.497,Z 423.016,A -85,B 0,C 180,E1 -9297.247,E2 -9297.247} C_VEL
LIN {X 0,Y 437.58,Z 416.617,A -85,B 0,C 180,E1 -9298.151,E2 -9298.151} C_VEL
LIN {X 0,Y 434.042,Z 401.252,A -85,B 0,C 180,E1 -9300.553,E2 -9300.553} C_VEL
LIN {X 0,Y 432.388,Z 394.787,A -85,B 0,C 180,E1 -9301.614,E2 -9301.614} C_VEL
LIN {X 0,Y 432.338,Z 394.632,A -85,B 0,C 180,E1 -9304.678,E2 -9304.678} C_VEL
LIN {X 0,Y 432.325,Z 394.635,A -85,B 0,C 180,E1 -9308.152,E2 -9308.152} C_VEL
LIN {X 0,Y 432.306,Z 394.635,A -85,B 0,C 180,E1 -9311.801,E2 -9311.801} C_VEL
LIN {X 0,Y 432.334,Z 394.615,A -85,B 0,C 180,E1 -9314.348,E2 -9314.348} C_VEL
LIN {X 0,Y 432.31,Z 394.633,A -85,B 0,C 180,E1 -9317.018,E2 -9317.018} C_VEL
LIN {X 0,Y 432.291,Z 394.637,A -85,B 0,C 180,E1 -9319.828,E2 -9319.828} C_VEL
LIN {X 0,Y 432.302,Z 394.628,A -85,B 0,C 180,E1 -9323.021,E2 -9323.021} C_VEL
LIN {X 0,Y 432.336,Z 394.624,A -85,B 0,C 180,E1 -9326.002,E2 -9326.002} C_VEL
LIN {X 0,Y 432.349,Z 394.633,A -85,B 0,C 180,E1 -9329.49,E2 -9329.49} C_VEL
LIN {X 0,Y 432.323,Z 394.629,A -85,B 0,C 180,E1 -9331.872,E2 -9331.872} C_VEL
LIN {X 0,Y 432.329,Z 394.629,A -85,B 0,C 180,E1 -9334.997,E2 -9334.997} C_VEL
LIN {X 0,Y 432.362,Z 394.629,A -85,B 0,C 180,E1 -9338.046,E2 -9338.046} C_VEL
LIN {X 0,Y 432.385,Z 394.62,A -85,B 0,C 180,E1 -9341.029,E2 -9341.029} C_VEL
LIN {X 0,Y 432.393,Z 394.624,A -85,B 0,C 180,E1 -9343.96,E2 -9343.96} C_VEL
LIN {X 0,Y 432.458,Z 394.604,A -85,B 0,C 180,E1 -9347.803,E2 -9347.803} C_VEL
LIN {X 0,Y 432.45,Z 394.617,A -85,B 0,C 180,E1 -9351.589,E2 -9351.589} C_VEL
LIN {X 0,Y 432.555,Z 394.591,A -85,B 0,C 180,E1 -9354.406,E2 -9354.406} C_VEL
LIN {X 0,Y 432.599,Z 394.598,A -85,B 0,C 180,E1 -9358.138,E2 -9358.138} C_VEL
LIN {X 0,Y 432.624,Z 394.592,A -85,B 0,C 180,E1 -9360,E2 -9360} C_VEL
LIN {X 0,Y 432.56,Z 394.585,A -85,B 0,C 180,E1 -9362.794,E2 -9362.794} C_VEL
LIN {X 0,Y 432.574,Z 394.601,A -85,B 0,C 180,E1 -9365.594,E2 -9365.594} C_VEL
LIN {X 0,Y 432.45,Z 394.605,A -85,B 0,C 180,E1 -9368.41,E2 -9368.41} C_VEL
LIN {X 0,Y 432.458,Z 394.615,A -85,B 0,C 180,E1 -9372.197,E2 -9372.197} C_VEL
LIN {X 0,Y 432.359,Z 394.614,A -85,B 0,C 180,E1 -9376.042,E2 -9376.042} C_VEL
LIN {X 0,Y 432.345,Z 394.629,A -85,B 0,C 180,E1 -9379.468,E2 -9379.468} C_VEL
LIN {X 0,Y 432.343,Z 394.62,A -85,B 0,C 180,E1 -9382.093,E2 -9382.093} C_VEL
LIN {X 0,Y 432.319,Z 394.628,A -85,B 0,C 180,E1 -9385.003,E2 -9385.003} C_VEL
LIN {X 0,Y 432.34,Z 394.617,A -85,B 0,C 180,E1 -9388.62,E2 -9388.62} C_VEL
LIN {X 0,Y 432.319,Z 394.631,A -85,B 0,C 180,E1 -9391.346,E2 -9391.346} C_VEL
LIN {X 0,Y 432.327,Z 394.622,A -85,B 0,C 180,E1 -9394.678,E2 -9394.678} C_VEL
LIN {X 0,Y 432.32,Z 394.628,A -85,B 0,C 180,E1 -9398.152,E2 -9398.152} C_VEL
LIN {X 0,Y 432.302,Z 394.604,A -85,B 0,C 180,E1 -9401.801,E2 -9401.801} C_VEL
LIN {X 0,Y 432.333,Z 394.631,A -85,B 0,C 180,E1 -9404.348,E2 -9404.348} C_VEL
LIN {X 0,Y 432.301,Z 394.629,A -85,B 0,C 180,E1 -9407.019,E2 -9407.019} C_VEL
LIN {X 0,Y 432.289,Z 394.616,A -85,B 0,C 180,E1 -9409.828,E2 -9409.828} C_VEL
LIN {X 0,Y 432.296,Z 394.635,A -85,B 0,C 180,E1 -9413.02,E2 -9413.02} C_VEL
LIN {X 0,Y 432.331,Z 394.635,A -85,B 0,C 180,E1 -9416.002,E2 -9416.002} C_VEL
LIN {X 0,Y 432.326,Z 394.807,A -85,B 0,C 180,E1 -9418.107,E2 -9418.107} C_VEL
LIN {X 0,Y 436.561,Z 412.884,A -85,B 0,C 180,E1 -9421.121,E2 -9421.121} C_VEL
LIN {X 0,Y 437.15,Z 416.473,A -85,B 0,C 180,E1 -9421.689,E2 -9421.689} C_VEL
LIN {X 0,Y 435.988,Z 436.48,A -85,B 0,C 180,E1 -9424.62,E2 -9424.62} C_VEL
LIN {X 0,Y 434.695,Z 459.283,A -85,B 0,C 180,E1 -9427.92,E2 -9427.92} C_VEL
LIN {X 0,Y 433.537,Z 484.416,A -85,B 0,C 180,E1 -9431.503,E2 -9431.503} C_VEL
LIN {X 0,Y 433.865,Z 488.826,A -85,B 0,C 180,E1 -9431.714,E2 -9431.714} C_VEL
LIN {X 0,Y 436.799,Z 516.585,A -85,B 0,C 180,E1 -9432.31,E2 -9432.31} C_VEL
LIN {X 0,Y 435.947,Z 607.351,A -85,B 0,C 180,E1 -9433.823,E2 -9433.823} C_VEL
LIN {X 0,Y 435.517,Z 620.41,A -85,B 0,C 180,E1 -9434.228,E2 -9434.228} C_VEL
LIN {X 0,Y 435.032,Z 633.523,A -85,B 0,C 180,E1 -9434.84,E2 -9434.84} C_VEL
LIN {X 0,Y 434.45,Z 645.315,A -85,B 0,C 180,E1 -9435.598,E2 -9435.598} C_VEL
LIN {X 0,Y 433.825,Z 656.55,A -85,B 0,C 180,E1 -9436.527,E2 -9436.527} C_VEL
LIN {X 0,Y 433.229,Z 666.778,A -85,B 0,C 180,E1 -9437.587,E2 -9437.587} C_VEL
LIN {X 0,Y 432.66,Z 675.881,A -85,B 0,C 180,E1 -9438.759,E2 -9438.759} C_VEL
LIN {X 0,Y 432.128,Z 684.722,A -85,B 0,C 180,E1 -9440.167,E2 -9440.167} C_VEL
LIN {X 0,Y 431.782,Z 691.803,A -85,B 0,C 180,E1 -9441.576,E2 -9441.576} C_VEL
LIN {X 0,Y 431.519,Z 697.425,A -85,B 0,C 180,E1 -9442.984,E2 -9442.984} C_VEL
LIN {X 0,Y 431.405,Z 701.827,A -85,B 0,C 180,E1 -9444.39,E2 -9444.39} C_VEL
LIN {X 0,Y 431.333,Z 704.143,A -85,B 0,C 180,E1 -9445.327,E2 -9445.327} C_VEL
LIN {X 0,Y 431.268,Z 706.029,A -85,B 0,C 180,E1 -9446.262,E2 -9446.262} C_VEL
LIN {X 0,Y 431.32,Z 707.453,A -85,B 0,C 180,E1 -9447.198,E2 -9447.198} C_VEL
LIN {X 0,Y 431.22,Z 709.07,A -85,B 0,C 180,E1 -9449.066,E2 -9449.066} C_VEL
LIN {X 0,Y 431.232,Z 709.289,A -85,B 0,C 180,E1 -9450,E2 -9450} C_VEL
LIN {X 0,Y 431.254,Z 709.069,A -85,B 0,C 180,E1 -9450.934,E2 -9450.934} C_VEL
LIN {X 0,Y 431.327,Z 707.452,A -85,B 0,C 180,E1 -9452.802,E2 -9452.802} C_VEL
LIN {X 0,Y 431.279,Z 706.026,A -85,B 0,C 180,E1 -9453.737,E2 -9453.737} C_VEL
LIN {X 0,Y 431.419,Z 703.059,A -85,B 0,C 180,E1 -9455.14,E2 -9455.14} C_VEL
LIN {X 0,Y 431.482,Z 699.027,A -85,B 0,C 180,E1 -9456.547,E2 -9456.547} C_VEL
LIN {X 0,Y 431.727,Z 692.803,A -85,B 0,C 180,E1 -9458.189,E2 -9458.189} C_VEL
LIN {X 0,Y 432.076,Z 686.007,A -85,B 0,C 180,E1 -9459.597,E2 -9459.597} C_VEL
LIN {X 0,Y 432.467,Z 679.046,A -85,B 0,C 180,E1 -9460.771,E2 -9460.771} C_VEL
LIN {X 0,Y 433.004,Z 670.627,A -85,B 0,C 180,E1 -9461.943,E2 -9461.943} C_VEL
LIN {X 0,Y 433.657,Z 660.193,A -85,B 0,C 180,E1 -9463.114,E2 -9463.114} C_VEL
LIN {X 0,Y 434.213,Z 649.841,A -85,B 0,C 180,E1 -9464.051,E2 -9464.051} C_VEL
LIN {X 0,Y 434.778,Z 638.408,A -85,B 0,C 180,E1 -9464.869,E2 -9464.869} C_VEL
LIN {X 0,Y 435.347,Z 626.51,A -85,B 0,C 180,E1 -9465.508,E2 -9465.508} C_VEL
LIN {X 0,Y 435.737,Z 613.619,A -85,B 0,C 180,E1 -9466.004,E2 -9466.004} C_VEL
LIN {X 0,Y 436.016,Z 601.421,A -85,B 0,C 180,E1 -9466.294,E2 -9466.294} C_VEL
LIN {X 0,Y 436.594,Z 548.046,A -85,B 0,C 180,E1 -9467.195,E2 -9467.195} C_VEL
LIN {X 0,Y 437.084,Z 514.485,A -85,B 0,C 180,E1 -9467.898,E2 -9467.898} C_VEL
LIN {X 0,Y 434.531,Z 486.529,A -85,B 0,C 180,E1 -9468.66,E2 -9468.66} C_VEL
LIN {X 0,Y 433.426,Z 477.939,A -85,B 0,C 180,E1 -9468.954,E2 -9468.954} C_VEL
LIN {X 0,Y 434.547,Z 454.783,A -85,B 0,C 180,E1 -9472.338,E2 -9472.338} C_VEL
LIN {X 0,Y 436.123,Z 430.415,A -85,B 0,C 180,E1 -9476.048,E2 -9476.048} C_VEL
LIN {X 0,Y 437.169,Z 416.221,A -85,B 0,C 180,E1 -9478.31,E2 -9478.31} C_VEL
LIN {X 0,Y 435.478,Z 407.016,A -85,B 0,C 180,E1 -9480.02,E2 -9480.02} C_VEL
LIN {X 0,Y 432.817,Z 396.598,A -85,B 0,C 180,E1 -9482.166,E2 -9482.166} C_VEL
LIN {X 0,Y 432.33,Z 394.691,A -85,B 0,C 180,E1 -9482.65,E2 -9482.65} C_VEL
LIN {X 0,Y 432.331,Z 394.635,A -85,B 0,C 180,E1 -9485.819,E2 -9485.819} C_VEL
LIN {X 0,Y 432.299,Z 394.637,A -85,B 0,C 180,E1 -9489.348,E2 -9489.348} C_VEL
LIN {X 0,Y 432.301,Z 394.637,A -85,B 0,C 180,E1 -9491.801,E2 -9491.801} C_VEL
LIN {X 0,Y 432.332,Z 394.632,A -85,B 0,C 180,E1 -9494.348,E2 -9494.348} C_VEL
LIN {X 0,Y 432.303,Z 394.633,A -85,B 0,C 180,E1 -9497.018,E2 -9497.018} C_VEL
LIN {X 0,Y 432.289,Z 394.637,A -85,B 0,C 180,E1 -9499.828,E2 -9499.828} C_VEL
LIN {X 0,Y 432.3,Z 394.636,A -85,B 0,C 180,E1 -9503.021,E2 -9503.021} C_VEL
LIN {X 0,Y 432.359,Z 394.629,A -85,B 0,C 180,E1 -9505.997,E2 -9505.997} C_VEL
LIN {X 0,Y 432.348,Z 394.63,A -85,B 0,C 180,E1 -9509.49,E2 -9509.49} C_VEL
LIN {X 0,Y 432.349,Z 394.632,A -85,B 0,C 180,E1 -9511.874,E2 -9511.874} C_VEL
LIN {X 0,Y 432.379,Z 394.627,A -85,B 0,C 180,E1 -9515.539,E2 -9515.539} C_VEL
LIN {X 0,Y 432.353,Z 394.632,A -85,B 0,C 180,E1 -9519.046,E2 -9519.046} C_VEL
LIN {X 0,Y 432.413,Z 394.85,A -85,B 0,C 180,E1 -9521.399,E2 -9521.399} C_VEL
LIN {X 0,Y 432.622,Z 395.748,A -85,B 0,C 180,E1 -9521.542,E2 -9521.542} C_VEL
LIN {X 0,Y 437.956,Z 407.938,A -85,B 0,C 180,E1 -9522.184,E2 -9522.184} C_VEL
LIN {X 0,Y 438.425,Z 410.307,A -85,B 0,C 180,E1 -9522.268,E2 -9522.268} C_VEL
LIN {X 0,Y 437.072,Z 478.961,A -85,B 0,C 180,E1 -9523.746,E2 -9523.746} C_VEL
LIN {X 0,Y 437.006,Z 491.771,A -85,B 0,C 180,E1 -9524.166,E2 -9524.166} C_VEL
LIN {X 0,Y 436.762,Z 504.188,A -85,B 0,C 180,E1 -9524.759,E2 -9524.759} C_VEL
LIN {X 0,Y 436.434,Z 516.324,A -85,B 0,C 180,E1 -9525.531,E2 -9525.531} C_VEL
LIN {X 0,Y 435.912,Z 527.806,A -85,B 0,C 180,E1 -9526.48,E2 -9526.48} C_VEL
LIN {X 0,Y 435.362,Z 537.959,A -85,B 0,C 180,E1 -9527.531,E2 -9527.531} C_VEL
LIN {X 0,Y 434.928,Z 546.223,A -85,B 0,C 180,E1 -9528.583,E2 -9528.583} C_VEL
LIN {X 0,Y 434.375,Z 553.818,A -85,B 0,C 180,E1 -9529.748,E2 -9529.748} C_VEL
LIN {X 0,Y 433.982,Z 560.717,A -85,B 0,C 180,E1 -9531.06,E2 -9531.06} C_VEL
LIN {X 0,Y 433.467,Z 566.979,A -85,B 0,C 180,E1 -9532.547,E2 -9532.547} C_VEL
LIN {X 0,Y 433.157,Z 571.543,A -85,B 0,C 180,E1 -9533.946,E2 -9533.946} C_VEL
LIN {X 0,Y 432.786,Z 574.982,A -85,B 0,C 180,E1 -9535.343,E2 -9535.343} C_VEL
LIN {X 0,Y 432.767,Z 576.674,A -85,B 0,C 180,E1 -9536.276,E2 -9536.276} C_VEL
LIN {X 0,Y 432.6,Z 577.91,A -85,B 0,C 180,E1 -9537.206,E2 -9537.206} C_VEL
LIN {X 0,Y 432.483,Z 578.731,A -85,B 0,C 180,E1 -9538.138,E2 -9538.138} C_VEL
LIN {X 0,Y 432.374,Z 579.152,A -85,B 0,C 180,E1 -9539.069,E2 -9539.069} C_VEL
LIN {X 0,Y 432.318,Z 579.119,A -85,B 0,C 180,E1 -9540,E2 -9540} C_VEL
LIN {X 0,Y 432.334,Z 578.659,A -85,B 0,C 180,E1 -9540.931,E2 -9540.931} C_VEL
LIN {X 0,Y 432.255,Z 577.816,A -85,B 0,C 180,E1 -9541.864,E2 -9541.864} C_VEL
LIN {X 0,Y 432.382,Z 576.526,A -85,B 0,C 180,E1 -9542.795,E2 -9542.795} C_VEL
LIN {X 0,Y 432.362,Z 573.794,A -85,B 0,C 180,E1 -9544.195,E2 -9544.195} C_VEL
LIN {X 0,Y 432.565,Z 569.995,A -85,B 0,C 180,E1 -9545.594,E2 -9545.594} C_VEL
LIN {X 0,Y 432.867,Z 565.037,A -85,B 0,C 180,E1 -9546.994,E2 -9546.994} C_VEL
LIN {X 0,Y 433.113,Z 558.789,A -85,B 0,C 180,E1 -9548.398,E2 -9548.398} C_VEL
LIN {X 0,Y 433.469,Z 551.014,A -85,B 0,C 180,E1 -9549.802,E2 -9549.802} C_VEL
LIN {X 0,Y 433.824,Z 543.07,A -85,B 0,C 180,E1 -9550.973,E2 -9550.973} C_VEL
LIN {X 0,Y 434.233,Z 533.356,A -85,B 0,C 180,E1 -9552.146,E2 -9552.146} C_VEL
LIN {X 0,Y 434.664,Z 522.565,A -85,B 0,C 180,E1 -9553.202,E2 -9553.202} C_VEL
LIN {X 0,Y 435.044,Z 510.673,A -85,B 0,C 180,E1 -9554.132,E2 -9554.132} C_VEL
LIN {X 0,Y 435.328,Z 497.773,A -85,B 0,C 180,E1 -9554.904,E2 -9554.904} C_VEL
LIN {X 0,Y 435.568,Z 484.919,A -85,B 0,C 180,E1 -9555.47,E2 -9555.47} C_VEL
LIN {X 0,Y 435.655,Z 471.616,A -85,B 0,C 180,E1 -9555.857,E2 -9555.857} C_VEL
LIN {X 0,Y 436.377,Z 407.027,A -85,B 0,C 180,E1 -9557.108,E2 -9557.108} C_VEL
LIN {X 0,Y 432.59,Z 395.618,A -85,B 0,C 180,E1 -9557.486,E2 -9557.486} C_VEL
LIN {X 0,Y 432.397,Z 394.709,A -85,B 0,C 180,E1 -9557.669,E2 -9557.669} C_VEL
LIN {X 0,Y 432.353,Z 394.632,A -85,B 0,C 180,E1 -9560.954,E2 -9560.954} C_VEL
LIN {X 0,Y 432.383,Z 394.627,A -85,B 0,C 180,E1 -9564.462,E2 -9564.462} C_VEL
LIN {X 0,Y 432.35,Z 394.622,A -85,B 0,C 180,E1 -9568.126,E2 -9568.126} C_VEL
LIN {X 0,Y 432.323,Z 394.632,A -85,B 0,C 180,E1 -9571.346,E2 -9571.346} C_VEL
LIN {X 0,Y 432.339,Z 394.625,A -85,B 0,C 180,E1 -9574.677,E2 -9574.677} C_VEL
LIN {X 0,Y 432.338,Z 394.625,A -85,B 0,C 180,E1 -9578.15,E2 -9578.15} C_VEL
LIN {X 0,Y 432.326,Z 394.627,A -85,B 0,C 180,E1 -9581.601,E2 -9581.601} C_VEL
LIN {X 0,Y 432.335,Z 394.634,A -85,B 0,C 180,E1 -9584.347,E2 -9584.347} C_VEL
LIN {X 0,Y 432.318,Z 394.632,A -85,B 0,C 180,E1 -9587.016,E2 -9587.016} C_VEL
LIN {X 0,Y 432.315,Z 394.633,A -85,B 0,C 180,E1 -9589.824,E2 -9589.824} C_VEL
LIN {X 0,Y 432.307,Z 394.637,A -85,B 0,C 180,E1 -9593.022,E2 -9593.022} C_VEL
LIN {X 0,Y 432.361,Z 394.627,A -85,B 0,C 180,E1 -9595.997,E2 -9595.997} C_VEL
LIN {X 0,Y 432.366,Z 394.799,A -85,B 0,C 180,E1 -9598.487,E2 -9598.487} C_VEL
LIN {X 0,Y 435.964,Z 409.337,A -85,B 0,C 180,E1 -9600.814,E2 -9600.814} C_VEL
LIN {X 0,Y 437.643,Z 417.112,A -85,B 0,C 180,E1 -9602.035,E2 -9602.035} C_VEL
LIN {X 0,Y 436.703,Z 438.43,A -85,B 0,C 180,E1 -9605.011,E2 -9605.011} C_VEL
LIN {X 0,Y 435.684,Z 459.864,A -85,B 0,C 180,E1 -9607.973,E2 -9607.973} C_VEL
LIN {X 0,Y 434.823,Z 481.86,A -85,B 0,C 180,E1 -9610.895,E2 -9610.895} C_VEL
LIN {X 0,Y 434.744,Z 487.83,A -85,B 0,C 180,E1 -9611.637,E2 -9611.637} C_VEL
LIN {X 0,Y 437.422,Z 506.921,A -85,B 0,C 180,E1 -9612.092,E2 -9612.092} C_VEL
LIN {X 0,Y 437.257,Z 521.92,A -85,B 0,C 180,E1 -9612.34,E2 -9612.34} C_VEL
LIN {X 0,Y 436.549,Z 527.766,A -85,B 0,C 180,E1 -9612.41,E2 -9612.41} C_VEL
LIN {X 0,Y 430.938,Z 546.783,A -85,B 0,C 180,E1 -9612.501,E2 -9612.501} C_VEL
LIN {X 0,Y 430.265,Z 552.628,A -85,B 0,C 180,E1 -9612.574,E2 -9612.574} C_VEL
LIN {X 0,Y 429.654,Z 600.069,A -85,B 0,C 180,E1 -9613.397,E2 -9613.397} C_VEL
LIN {X 0,Y 429.193,Z 613.041,A -85,B 0,C 180,E1 -9613.806,E2 -9613.806} C_VEL
LIN {X 0,Y 428.63,Z 625.981,A -85,B 0,C 180,E1 -9614.426,E2 -9614.426} C_VEL
LIN {X 0,Y 428.04,Z 637.057,A -85,B 0,C 180,E1 -9615.135,E2 -9615.135} C_VEL
LIN {X 0,Y 427.391,Z 648.009,A -85,B 0,C 180,E1 -9616.032,E2 -9616.032} C_VEL
LIN {X 0,Y 426.784,Z 657.802,A -85,B 0,C 180,E1 -9617.034,E2 -9617.034} C_VEL
LIN {X 0,Y 426.031,Z 668.153,A -85,B 0,C 180,E1 -9618.341,E2 -9618.341} C_VEL
LIN {X 0,Y 425.384,Z 677.139,A -85,B 0,C 180,E1 -9619.77,E2 -9619.77} C_VEL
LIN {X 0,Y 424.922,Z 684.352,A -85,B 0,C 180,E1 -9621.2,E2 -9621.2} C_VEL
LIN {X 0,Y 424.546,Z 690.975,A -85,B 0,C 180,E1 -9622.868,E2 -9622.868} C_VEL
LIN {X 0,Y 424.368,Z 695.326,A -85,B 0,C 180,E1 -9624.297,E2 -9624.297} C_VEL
LIN {X 0,Y 424.244,Z 697.616,A -85,B 0,C 180,E1 -9625.249,E2 -9625.249} C_VEL
LIN {X 0,Y 424.124,Z 699.485,A -85,B 0,C 180,E1 -9626.2,E2 -9626.2} C_VEL
LIN {X 0,Y 424.141,Z 700.914,A -85,B 0,C 180,E1 -9627.151,E2 -9627.151} C_VEL
LIN {X 0,Y 424.13,Z 701.914,A -85,B 0,C 180,E1 -9628.101,E2 -9628.101} C_VEL
LIN {X 0,Y 424.062,Z 702.77,A -85,B 0,C 180,E1 -9630,E2 -9630} C_VEL
LIN {X 0,Y 424.07,Z 702.579,A -85,B 0,C 180,E1 -9630.95,E2 -9630.95} C_VEL
LIN {X 0,Y 424.13,Z 701.991,A -85,B 0,C 180,E1 -9631.899,E2 -9631.899} C_VEL
LIN {X 0,Y 424.141,Z 701.021,A -85,B 0,C 180,E1 -9632.849,E2 -9632.849} C_VEL
LIN {X 0,Y 424.124,Z 699.651,A -85,B 0,C 180,E1 -9633.801,E2 -9633.801} C_VEL
LIN {X 0,Y 424.301,Z 696.771,A -85,B 0,C 180,E1 -9635.227,E2 -9635.227} C_VEL
LIN {X 0,Y 424.401,Z 692.858,A -85,B 0,C 180,E1 -9636.657,E2 -9636.657} C_VEL
LIN {X 0,Y 424.684,Z 687.79,A -85,B 0,C 180,E1 -9638.086,E2 -9638.086} C_VEL
LIN {X 0,Y 425.086,Z 681.402,A -85,B 0,C 180,E1 -9639.517,E2 -9639.517} C_VEL
LIN {X 0,Y 425.642,Z 673.469,A -85,B 0,C 180,E1 -9640.946,E2 -9640.946} C_VEL
LIN {X 0,Y 426.256,Z 665.366,A -85,B 0,C 180,E1 -9642.135,E2 -9642.135} C_VEL
LIN {X 0,Y 427.023,Z 655.415,A -85,B 0,C 180,E1 -9643.322,E2 -9643.322} C_VEL
LIN {X 0,Y 427.491,Z 645.608,A -85,B 0,C 180,E1 -9644.277,E2 -9644.277} C_VEL
LIN {X 0,Y 428.168,Z 634.989,A -85,B 0,C 180,E1 -9645.104,E2 -9645.104} C_VEL
LIN {X 0,Y 428.795,Z 623.369,A -85,B 0,C 180,E1 -9645.812,E2 -9645.812} C_VEL
LIN {X 0,Y 429.312,Z 610.757,A -85,B 0,C 180,E1 -9646.373,E2 -9646.373} C_VEL
LIN {X 0,Y 429.722,Z 597.599,A -85,B 0,C 180,E1 -9646.754,E2 -9646.754} C_VEL
LIN {X 0,Y 430.526,Z 506.498,A -85,B 0,C 180,E1 -9648.306,E2 -9648.306} C_VEL
LIN {X 0,Y 427.866,Z 487.672,A -85,B 0,C 180,E1 -9648.777,E2 -9648.777} C_VEL
LIN {X 0,Y 428.56,Z 467.683,A -85,B 0,C 180,E1 -9651.4,E2 -9651.4} C_VEL
LIN {X 0,Y 429.653,Z 444.189,A -85,B 0,C 180,E1 -9654.653,E2 -9654.653} C_VEL
LIN {X 0,Y 430.709,Z 424.364,A -85,B 0,C 180,E1 -9657.45,E2 -9657.45} C_VEL
LIN {X 0,Y 430.84,Z 418.716,A -85,B 0,C 180,E1 -9658.253,E2 -9658.253} C_VEL
LIN {X 0,Y 427.391,Z 403.548,A -85,B 0,C 180,E1 -9660.648,E2 -9660.648} C_VEL
LIN {X 0,Y 425.337,Z 395.632,A -85,B 0,C 180,E1 -9661.976,E2 -9661.976} C_VEL
LIN {X 0,Y 425.298,Z 395.514,A -85,B 0,C 180,E1 -9665.336,E2 -9665.336} C_VEL
LIN {X 0,Y 425.279,Z 395.512,A -85,B 0,C 180,E1 -9668.901,E2 -9668.901} C_VEL
LIN {X 0,Y 425.259,Z 395.512,A -85,B 0,C 180,E1 -9672.656,E2 -9672.656} C_VEL
LIN {X 0,Y 425.286,Z 395.492,A -85,B 0,C 180,E1 -9675.283,E2 -9675.283} C_VEL
LIN {X 0,Y 425.253,Z 395.511,A -85,B 0,C 180,E1 -9678.619,E2 -9678.619} C_VEL
LIN {X 0,Y 425.281,Z 395.51,A -85,B 0,C 180,E1 -9681.099,E2 -9681.099} C_VEL
LIN {X 0,Y 425.297,Z 395.506,A -85,B 0,C 180,E1 -9684.664,E2 -9684.664} C_VEL
LIN {X 0,Y 425.267,Z 395.513,A -85,B 0,C 180,E1 -9688.073,E2 -9688.073} C_VEL
LIN {X 0,Y 425.3,Z 395.5,A -85,B 0,C 180,E1 -9691.365,E2 -9691.365} C_VEL
LIN {X 0,Y 425.265,Z 395.509,A -85,B 0,C 180,E1 -9694.553,E2 -9694.553} C_VEL
LIN {X 0,Y 425.296,Z 395.504,A -85,B 0,C 180,E1 -9697.73,E2 -9697.73} C_VEL
LIN {X 0,Y 425.364,Z 395.494,A -85,B 0,C 180,E1 -9700.704,E2 -9700.704} C_VEL
LIN {X 0,Y 425.327,Z 395.499,A -85,B 0,C 180,E1 -9703.686,E2 -9703.686} C_VEL
LIN {X 0,Y 425.397,Z 395.491,A -85,B 0,C 180,E1 -9707.097,E2 -9707.097} C_VEL
LIN {X 0,Y 425.385,Z 395.492,A -85,B 0,C 180,E1 -9710.49,E2 -9710.49} C_VEL
LIN {X 0,Y 425.48,Z 395.484,A -85,B 0,C 180,E1 -9713.36,E2 -9713.36} C_VEL
LIN {X 0,Y 425.346,Z 395.488,A -85,B 0,C 180,E1 -9715.261,E2 -9715.261} C_VEL
LIN {X 0,Y 425.568,Z 395.474,A -85,B 0,C 180,E1 -9718.107,E2 -9718.107} C_VEL
LIN {X 0,Y 425.576,Z 395.47,A -85,B 0,C 180,E1 -9720,E2 -9720} C_VEL
LIN {X 0,Y 425.516,Z 395.462,A -85,B 0,C 180,E1 -9722.84,E2 -9722.84} C_VEL
LIN {X 0,Y 425.528,Z 395.48,A -85,B 0,C 180,E1 -9725.687,E2 -9725.687} C_VEL
LIN {X 0,Y 425.398,Z 395.483,A -85,B 0,C 180,E1 -9728.551,E2 -9728.551} C_VEL
LIN {X 0,Y 425.412,Z 395.491,A -85,B 0,C 180,E1 -9732.402,E2 -9732.402} C_VEL
LIN {X 0,Y 425.311,Z 395.49,A -85,B 0,C 180,E1 -9736.315,E2 -9736.315} C_VEL
LIN {X 0,Y 425.295,Z 395.509,A -85,B 0,C 180,E1 -9739.621,E2 -9739.621} C_VEL
LIN {X 0,Y 425.289,Z 395.496,A -85,B 0,C 180,E1 -9742.339,E2 -9742.339} C_VEL
LIN {X 0,Y 425.254,Z 395.511,A -85,B 0,C 180,E1 -9745.448,E2 -9745.448} C_VEL
LIN {X 0,Y 425.303,Z 395.493,A -85,B 0,C 180,E1 -9748.858,E2 -9748.858} C_VEL
LIN {X 0,Y 425.265,Z 395.514,A -85,B 0,C 180,E1 -9751.927,E2 -9751.927} C_VEL
LIN {X 0,Y 425.294,Z 395.5,A -85,B 0,C 180,E1 -9755.337,E2 -9755.337} C_VEL
LIN {X 0,Y 425.267,Z 395.503,A -85,B 0,C 180,E1 -9758.902,E2 -9758.902} C_VEL
LIN {X 0,Y 425.264,Z 395.48,A -85,B 0,C 180,E1 -9761.954,E2 -9761.954} C_VEL
LIN {X 0,Y 425.285,Z 395.508,A -85,B 0,C 180,E1 -9765.283,E2 -9765.283} C_VEL
LIN {X 0,Y 425.246,Z 395.486,A -85,B 0,C 180,E1 -9768.618,E2 -9768.618} C_VEL
LIN {X 0,Y 425.27,Z 395.513,A -85,B 0,C 180,E1 -9772.304,E2 -9772.304} C_VEL
LIN {X 0,Y 425.284,Z 395.513,A -85,B 0,C 180,E1 -9775.815,E2 -9775.815} C_VEL
LIN {X 0,Y 425.32,Z 395.71,A -85,B 0,C 180,E1 -9777.86,E2 -9777.86} C_VEL
LIN {X 0,Y 429.828,Z 415.275,A -85,B 0,C 180,E1 -9781.161,E2 -9781.161} C_VEL
LIN {X 0,Y 430.205,Z 420.015,A -85,B 0,C 180,E1 -9781.905,E2 -9781.905} C_VEL
LIN {X 0,Y 428.773,Z 441.105,A -85,B 0,C 180,E1 -9785.035,E2 -9785.035} C_VEL
LIN {X 0,Y 427.482,Z 463.29,A -85,B 0,C 180,E1 -9788.29,E2 -9788.29} C_VEL
LIN {X 0,Y 426.536,Z 482.648,A -85,B 0,C 180,E1 -9791.102,E2 -9791.102} C_VEL
LIN {X 0,Y 426.958,Z 488.182,A -85,B 0,C 180,E1 -9791.391,E2 -9791.391} C_VEL
LIN {X 0,Y 430.049,Z 516.893,A -85,B 0,C 180,E1 -9792.026,E2 -9792.026} C_VEL
LIN {X 0,Y 429.147,Z 607.384,A -85,B 0,C 180,E1 -9793.56,E2 -9793.56} C_VEL
LIN {X 0,Y 428.691,Z 620.408,A -85,B 0,C 180,E1 -9793.97,E2 -9793.97} C_VEL
LIN {X 0,Y 428.176,Z 633.502,A -85,B 0,C 180,E1 -9794.591,E2 -9794.591} C_VEL
LIN {X 0,Y 427.571,Z 645.283,A -85,B 0,C 180,E1 -9795.361,E2 -9795.361} C_VEL
LIN {X 0,Y 426.941,Z 656.194,A -85,B 0,C 180,E1 -9796.276,E2 -9796.276} C_VEL
LIN {X 0,Y 426.294,Z 666.735,A -85,B 0,C 180,E1 -9797.382,E2 -9797.382} C_VEL
LIN {X 0,Y 425.673,Z 675.835,A -85,B 0,C 180,E1 -9798.573,E2 -9798.573} C_VEL
LIN {X 0,Y 425.096,Z 684.674,A -85,B 0,C 180,E1 -9800.003,E2 -9800.003} C_VEL
LIN {X 0,Y 424.723,Z 691.753,A -85,B 0,C 180,E1 -9801.435,E2 -9801.435} C_VEL
LIN {X 0,Y 424.438,Z 697.374,A -85,B 0,C 180,E1 -9802.866,E2 -9802.866} C_VEL
LIN {X 0,Y 424.303,Z 701.775,A -85,B 0,C 180,E1 -9804.296,E2 -9804.296} C_VEL
LIN {X 0,Y 424.267,Z 704.09,A -85,B 0,C 180,E1 -9805.249,E2 -9805.249} C_VEL
LIN {X 0,Y 424.175,Z 705.976,A -85,B 0,C 180,E1 -9806.2,E2 -9806.2} C_VEL
LIN {X 0,Y 424.215,Z 707.4,A -85,B 0,C 180,E1 -9807.151,E2 -9807.151} C_VEL
LIN {X 0,Y 424.185,Z 708.403,A -85,B 0,C 180,E1 -9808.101,E2 -9808.101} C_VEL
LIN {X 0,Y 424.146,Z 709.235,A -85,B 0,C 180,E1 -9810,E2 -9810} C_VEL
LIN {X 0,Y 424.169,Z 709.015,A -85,B 0,C 180,E1 -9810.949,E2 -9810.949} C_VEL
LIN {X 0,Y 424.189,Z 708.401,A -85,B 0,C 180,E1 -9811.899,E2 -9811.899} C_VEL
LIN {X 0,Y 424.222,Z 707.397,A -85,B 0,C 180,E1 -9812.849,E2 -9812.849} C_VEL
LIN {X 0,Y 424.186,Z 705.972,A -85,B 0,C 180,E1 -9813.8,E2 -9813.8} C_VEL
LIN {X 0,Y 424.329,Z 703.005,A -85,B 0,C 180,E1 -9815.226,E2 -9815.226} C_VEL
LIN {X 0,Y 424.399,Z 698.973,A -85,B 0,C 180,E1 -9816.657,E2 -9816.657} C_VEL
LIN {X 0,Y 424.694,Z 692.75,A -85,B 0,C 180,E1 -9818.326,E2 -9818.326} C_VEL
LIN {X 0,Y 425.059,Z 685.955,A -85,B 0,C 180,E1 -9819.757,E2 -9819.757} C_VEL
LIN {X 0,Y 425.455,Z 678.995,A -85,B 0,C 180,E1 -9820.951,E2 -9820.951} C_VEL
LIN {X 0,Y 426.044,Z 670.578,A -85,B 0,C 180,E1 -9822.141,E2 -9822.141} C_VEL
LIN {X 0,Y 426.725,Z 660.148,A -85,B 0,C 180,E1 -9823.331,E2 -9823.331} C_VEL
LIN {X 0,Y 427.321,Z 649.799,A -85,B 0,C 180,E1 -9824.282,E2 -9824.282} C_VEL
LIN {X 0,Y 427.925,Z 638.373,A -85,B 0,C 180,E1 -9825.113,E2 -9825.113} C_VEL
LIN {X 0,Y 428.526,Z 626.486,A -85,B 0,C 180,E1 -9825.761,E2 -9825.761} C_VEL
LIN {X 0,Y 428.933,Z 613.613,A -85,B 0,C 180,E1 -9826.265,E2 -9826.265} C_VEL
LIN {X 0,Y 429.208,Z 601.468,A -85,B 0,C 180,E1 -9826.56,E2 -9826.56} C_VEL
LIN {X 0,Y 429.755,Z 555.365,A -85,B 0,C 180,E1 -9827.355,E2 -9827.355} C_VEL
LIN {X 0,Y 430.449,Z 514.868,A -85,B 0,C 180,E1 -9828.225,E2 -9828.225} C_VEL
LIN {X 0,Y 427.911,Z 486.881,A -85,B 0,C 180,E1 -9829.023,E2 -9829.023} C_VEL
LIN {X 0,Y 426.529,Z 476.534,A -85,B 0,C 180,E1 -9829.388,E2 -9829.388} C_VEL
LIN {X 0,Y 427.847,Z 451.834,A -85,B 0,C 180,E1 -9833.091,E2 -9833.091} C_VEL
LIN {X 0,Y 429.382,Z 430.175,A -85,B 0,C 180,E1 -9836.489,E2 -9836.489} C_VEL
LIN {X 0,Y 430.375,Z 417.716,A -85,B 0,C 180,E1 -9838.532,E2 -9838.532} C_VEL
LIN {X 0,Y 428.631,Z 408.436,A -85,B 0,C 180,E1 -9840.317,E2 -9840.317} C_VEL
LIN {X 0,Y 425.809,Z 397.467,A -85,B 0,C 180,E1 -9842.674,E2 -9842.674} C_VEL
LIN {X 0,Y 425.283,Z 395.568,A -85,B 0,C 180,E1 -9843.189,E2 -9843.189} C_VEL
LIN {X 0,Y 425.256,Z 395.516,A -85,B 0,C 180,E1 -9846.509,E2 -9846.509} C_VEL
LIN {X 0,Y 425.256,Z 395.515,A -85,B 0,C 180,E1 -9849.036,E2 -9849.036} C_VEL
LIN {X 0,Y 425.256,Z 395.514,A -85,B 0,C 180,E1 -9852.656,E2 -9852.656} C_VEL
LIN {X 0,Y 425.284,Z 395.509,A -85,B 0,C 180,E1 -9855.283,E2 -9855.283} C_VEL
LIN {X 0,Y 425.248,Z 395.512,A -85,B 0,C 180,E1 -9858.618,E2 -9858.618} C_VEL
LIN {X 0,Y 425.279,Z 395.511,A -85,B 0,C 180,E1 -9861.099,E2 -9861.099} C_VEL
LIN {X 0,Y 425.298,Z 395.508,A -85,B 0,C 180,E1 -9864.664,E2 -9864.664} C_VEL
LIN {X 0,Y 425.267,Z 395.513,A -85,B 0,C 180,E1 -9868.073,E2 -9868.073} C_VEL
LIN {X 0,Y 425.316,Z 395.506,A -85,B 0,C 180,E1 -9871.367,E2 -9871.367} C_VEL
LIN {X 0,Y 425.273,Z 395.51,A -85,B 0,C 180,E1 -9874.553,E2 -9874.553} C_VEL
LIN {X 0,Y 425.306,Z 395.509,A -85,B 0,C 180,E1 -9876.635,E2 -9876.635} C_VEL
LIN {X 0,Y 425.331,Z 395.506,A -85,B 0,C 180,E1 -9880.364,E2 -9880.364} C_VEL
LIN {X 0,Y 425.385,Z 395.751,A -85,B 0,C 180,E1 -9880.955,E2 -9880.955} C_VEL
LIN {X 0,Y 425.662,Z 396.873,A -85,B 0,C 180,E1 -9881.112,E2 -9881.112} C_VEL
LIN {X 0,Y 431.482,Z 409.812,A -85,B 0,C 180,E1 -9881.831,E2 -9881.831} C_VEL
LIN {X 0,Y 431.922,Z 411.342,A -85,B 0,C 180,E1 -9881.897,E2 -9881.897} C_VEL
LIN {X 0,Y 430.471,Z 478.91,A -85,B 0,C 180,E1 -9883.399,E2 -9883.399} C_VEL
LIN {X 0,Y 430.397,Z 492.131,A -85,B 0,C 180,E1 -9883.822,E2 -9883.822} C_VEL
LIN {X 0,Y 430.169,Z 504.453,A -85,B 0,C 180,E1 -9884.41,E2 -9884.41} C_VEL
LIN {X 0,Y 429.794,Z 516.358,A -85,B 0,C 180,E1 -9885.168,E2 -9885.168} C_VEL
LIN {X 0,Y 429.321,Z 526.949,A -85,B 0,C 180,E1 -9886.027,E2 -9886.027} C_VEL
LIN {X 0,Y 428.788,Z 536.378,A -85,B 0,C 180,E1 -9886.975,E2 -9886.975} C_VEL
LIN {X 0,Y 428.196,Z 545.989,A -85,B 0,C 180,E1 -9888.161,E2 -9888.161} C_VEL
LIN {X 0,Y 427.653,Z 553.829,A -85,B 0,C 180,E1 -9889.346,E2 -9889.346} C_VEL
LIN {X 0,Y 427.183,Z 560.277,A -85,B 0,C 180,E1 -9890.531,E2 -9890.531} C_VEL
LIN {X 0,Y 426.699,Z 566.559,A -85,B 0,C 180,E1 -9891.952,E2 -9891.952} C_VEL
LIN {X 0,Y 426.251,Z 571.474,A -85,B 0,C 180,E1 -9893.372,E2 -9893.372} C_VEL
LIN {X 0,Y 425.968,Z 575.19,A -85,B 0,C 180,E1 -9894.794,E2 -9894.794} C_VEL
LIN {X 0,Y 425.78,Z 577.837,A -85,B 0,C 180,E1 -9896.214,E2 -9896.214} C_VEL
LIN {X 0,Y 425.6,Z 579.043,A -85,B 0,C 180,E1 -9897.16,E2 -9897.16} C_VEL
LIN {X 0,Y 425.475,Z 579.84,A -85,B 0,C 180,E1 -9898.107,E2 -9898.107} C_VEL
LIN {X 0,Y 425.358,Z 580.232,A -85,B 0,C 180,E1 -9899.053,E2 -9899.053} C_VEL
LIN {X 0,Y 425.295,Z 580.159,A -85,B 0,C 180,E1 -9900,E2 -9900} C_VEL
LIN {X 0,Y 425.311,Z 579.665,A -85,B 0,C 180,E1 -9900.947,E2 -9900.947} C_VEL
LIN {X 0,Y 425.232,Z 578.789,A -85,B 0,C 180,E1 -9901.894,E2 -9901.894} C_VEL
LIN {X 0,Y 425.36,Z 577.445,A -85,B 0,C 180,E1 -9902.841,E2 -9902.841} C_VEL
LIN {X 0,Y 425.339,Z 574.645,A -85,B 0,C 180,E1 -9904.264,E2 -9904.264} C_VEL
LIN {X 0,Y 425.564,Z 570.767,A -85,B 0,C 180,E1 -9905.687,E2 -9905.687} C_VEL
LIN {X 0,Y 425.876,Z 565.724,A -85,B 0,C 180,E1 -9907.11,E2 -9907.11} C_VEL
LIN {X 0,Y 426.107,Z 559.383,A -85,B 0,C 180,E1 -9908.537,E2 -9908.537} C_VEL
LIN {X 0,Y 426.474,Z 551.489,A -85,B 0,C 180,E1 -9909.964,E2 -9909.964} C_VEL
LIN {X 0,Y 426.854,Z 543.402,A -85,B 0,C 180,E1 -9911.155,E2 -9911.155} C_VEL
LIN {X 0,Y 427.287,Z 533.511,A -85,B 0,C 180,E1 -9912.347,E2 -9912.347} C_VEL
LIN {X 0,Y 427.74,Z 522.538,A -85,B 0,C 180,E1 -9913.419,E2 -9913.419} C_VEL
LIN {X 0,Y 428.091,Z 510.831,A -85,B 0,C 180,E1 -9914.329,E2 -9914.329} C_VEL
LIN {X 0,Y 428.397,Z 498.043,A -85,B 0,C 180,E1 -9915.096,E2 -9915.096} C_VEL
LIN {X 0,Y 428.635,Z 485.012,A -85,B 0,C 180,E1 -9915.666,E2 -9915.666} C_VEL
LIN {X 0,Y 428.711,Z 471.276,A -85,B 0,C 180,E1 -9916.06,E2 -9916.06} C_VEL
LIN {X 0,Y 429.476,Z 408.325,A -85,B 0,C 180,E1 -9917.313,E2 -9917.313} C_VEL
LIN {X 0,Y 425.492,Z 396.297,A -85,B 0,C 180,E1 -9917.728,E2 -9917.728} C_VEL
LIN {X 0,Y 425.355,Z 395.571,A -85,B 0,C 180,E1 -9917.908,E2 -9917.908} C_VEL
LIN {X 0,Y 425.298,Z 395.51,A -85,B 0,C 180,E1 -9920.305,E2 -9920.305} C_VEL
LIN {X 0,Y 425.309,Z 395.506,A -85,B 0,C 180,E1 -9923.365,E2 -9923.365} C_VEL
LIN {X 0,Y 425.305,Z 395.509,A -85,B 0,C 180,E1 -9926.498,E2 -9926.498} C_VEL
LIN {X 0,Y 425.288,Z 395.501,A -85,B 0,C 180,E1 -9929.72,E2 -9929.72} C_VEL
LIN {X 0,Y 425.284,Z 395.501,A -85,B 0,C 180,E1 -9933.048,E2 -9933.048} C_VEL
LIN {X 0,Y 425.283,Z 395.507,A -85,B 0,C 180,E1 -9935.929,E2 -9935.929} C_VEL
LIN {X 0,Y 425.284,Z 395.508,A -85,B 0,C 180,E1 -9939.041,E2 -9939.041} C_VEL
LIN {X 0,Y 425.284,Z 395.504,A -85,B 0,C 180,E1 -9941.957,E2 -9941.957} C_VEL
LIN {X 0,Y 425.287,Z 395.505,A -85,B 0,C 180,E1 -9945.283,E2 -9945.283} C_VEL
LIN {X 0,Y 425.267,Z 395.512,A -85,B 0,C 180,E1 -9948.62,E2 -9948.62} C_VEL
LIN {X 0,Y 425.283,Z 395.495,A -85,B 0,C 180,E1 -9951.099,E2 -9951.099} C_VEL
LIN {X 0,Y 425.301,Z 395.498,A -85,B 0,C 180,E1 -9954.664,E2 -9954.664} C_VEL
LIN {X 0,Y 425.341,Z 395.671,A -85,B 0,C 180,E1 -9958.142,E2 -9958.142} C_VEL
LIN {X 0,Y 429.06,Z 410.535,A -85,B 0,C 180,E1 -9960.567,E2 -9960.567} C_VEL
LIN {X 0,Y 430.911,Z 419.621,A -85,B 0,C 180,E1 -9961.99,E2 -9961.99} C_VEL
LIN {X 0,Y 429.698,Z 443.444,A -85,B 0,C 180,E1 -9965.35,E2 -9965.35} C_VEL
LIN {X 0,Y 428.569,Z 466.958,A -85,B 0,C 180,E1 -9968.6,E2 -9968.6} C_VEL
LIN {X 0,Y 427.857,Z 487.83,A -85,B 0,C 180,E1 -9971.331,E2 -9971.331} C_VEL
LIN {X 0,Y 430.664,Z 507.861,A -85,B 0,C 180,E1 -9971.819,E2 -9971.819} C_VEL
LIN {X 0,Y 430.265,Z 552.628,A -85,B 0,C 180,E1 -9972.574,E2 -9972.574} C_VEL
LIN {X 0,Y 429.555,Z 558.477,A -85,B 0,C 180,E1 -9972.645,E2 -9972.645} C_VEL
LIN {X 0,Y 423.714,Z 577.457,A -85,B 0,C 180,E1 -9972.731,E2 -9972.731} C_VEL
LIN {X 0,Y 423.045,Z 583.304,A -85,B 0,C 180,E1 -9972.805,E2 -9972.805} C_VEL
LIN {X 0,Y 422.854,Z 601.33,A -85,B 0,C 180,E1 -9973.153,E2 -9973.153} C_VEL
LIN {X 0,Y 422.326,Z 614.472,A -85,B 0,C 180,E1 -9973.598,E2 -9973.598} C_VEL
LIN {X 0,Y 421.725,Z 627.082,A -85,B 0,C 180,E1 -9974.226,E2 -9974.226} C_VEL
LIN {X 0,Y 421.07,Z 638.707,A -85,B 0,C 180,E1 -9975.007,E2 -9975.007} C_VEL
LIN {X 0,Y 420.373,Z 650.585,A -85,B 0,C 180,E1 -9976.045,E2 -9976.045} C_VEL
LIN {X 0,Y 419.686,Z 660.936,A -85,B 0,C 180,E1 -9977.18,E2 -9977.18} C_VEL
LIN {X 0,Y 418.899,Z 669.834,A -85,B 0,C 180,E1 -9978.385,E2 -9978.385} C_VEL
LIN {X 0,Y 418.297,Z 678.513,A -85,B 0,C 180,E1 -9979.839,E2 -9979.839} C_VEL
LIN {X 0,Y 417.824,Z 685.485,A -85,B 0,C 180,E1 -9981.293,E2 -9981.293} C_VEL
LIN {X 0,Y 417.469,Z 691.029,A -85,B 0,C 180,E1 -9982.747,E2 -9982.747} C_VEL
LIN {X 0,Y 417.276,Z 695.38,A -85,B 0,C 180,E1 -9984.2,E2 -9984.2} C_VEL
LIN {X 0,Y 417.181,Z 697.67,A -85,B 0,C 180,E1 -9985.168,E2 -9985.168} C_VEL
LIN {X 0,Y 417.04,Z 699.539,A -85,B 0,C 180,E1 -9986.135,E2 -9986.135} C_VEL
LIN {X 0,Y 417.039,Z 700.968,A -85,B 0,C 180,E1 -9987.102,E2 -9987.102} C_VEL
LIN {X 0,Y 417.057,Z 701.969,A -85,B 0,C 180,E1 -9988.069,E2 -9988.069} C_VEL
LIN {X 0,Y 416.983,Z 702.824,A -85,B 0,C 180,E1 -9990,E2 -9990} C_VEL
LIN {X 0,Y 416.993,Z 702.633,A -85,B 0,C 180,E1 -9990.966,E2 -9990.966} C_VEL
LIN {X 0,Y 417.058,Z 702.044,A -85,B 0,C 180,E1 -9991.932,E2 -9991.932} C_VEL
LIN {X 0,Y 417.039,Z 701.074,A -85,B 0,C 180,E1 -9992.898,E2 -9992.898} C_VEL
LIN {X 0,Y 417.039,Z 699.704,A -85,B 0,C 180,E1 -9993.865,E2 -9993.865} C_VEL
LIN {X 0,Y 417.222,Z 696.823,A -85,B 0,C 180,E1 -9995.316,E2 -9995.316} C_VEL
LIN {X 0,Y 417.326,Z 692.909,A -85,B 0,C 180,E1 -9996.77,E2 -9996.77} C_VEL
LIN {X 0,Y 417.627,Z 687.84,A -85,B 0,C 180,E1 -9998.224,E2 -9998.224} C_VEL
LIN {X 0,Y 418.077,Z 681.45,A -85,B 0,C 180,E1 -9999.678,E2 -9999.678} C_VEL
LIN {X 0,Y 418.653,Z 673.515,A -85,B 0,C 180,E1 -10001.131,E2 -10001.131} C_VEL
LIN {X 0,Y 419.311,Z 665.41,A -85,B 0,C 180,E1 -10002.34,E2 -10002.34} C_VEL
LIN {X 0,Y 420.106,Z 655.454,A -85,B 0,C 180,E1 -10003.545,E2 -10003.545} C_VEL
LIN {X 0,Y 420.614,Z 645.642,A -85,B 0,C 180,E1 -10004.515,E2 -10004.515} C_VEL
LIN {X 0,Y 421.329,Z 635.016,A -85,B 0,C 180,E1 -10005.356,E2 -10005.356} C_VEL
LIN {X 0,Y 421.988,Z 623.385,A -85,B 0,C 180,E1 -10006.074,E2 -10006.074} C_VEL
LIN {X 0,Y 422.522,Z 610.748,A -85,B 0,C 180,E1 -10006.643,E2 -10006.643} C_VEL
LIN {X 0,Y 422.927,Z 597.546,A -85,B 0,C 180,E1 -10007.031,E2 -10007.031} C_VEL
LIN {X 0,Y 423.806,Z 507.318,A -85,B 0,C 180,E1 -10008.59,E2 -10008.59} C_VEL
LIN {X 0,Y 421.031,Z 487.862,A -85,B 0,C 180,E1 -10009.077,E2 -10009.077} C_VEL
LIN {X 0,Y 421.681,Z 469.336,A -85,B 0,C 180,E1 -10011.51,E2 -10011.51} C_VEL
LIN {X 0,Y 422.816,Z 445.649,A -85,B 0,C 180,E1 -10014.816,E2 -10014.816} C_VEL
LIN {X 0,Y 423.936,Z 425.738,A -85,B 0,C 180,E1 -10017.658,E2 -10017.658} C_VEL
LIN {X 0,Y 424.131,Z 421.263,A -85,B 0,C 180,E1 -10018.293,E2 -10018.293} C_VEL
LIN {X 0,Y 420.959,Z 406.749,A -85,B 0,C 180,E1 -10020.611,E2 -10020.611} C_VEL
LIN {X 0,Y 418.282,Z 396.581,A -85,B 0,C 180,E1 -10022.311,E2 -10022.311} C_VEL
LIN {X 0,Y 418.26,Z 396.387,A -85,B 0,C 180,E1 -10024.841,E2 -10024.841} C_VEL
LIN {X 0,Y 418.237,Z 396.389,A -85,B 0,C 180,E1 -10028.444,E2 -10028.444} C_VEL
LIN {X 0,Y 418.222,Z 396.39,A -85,B 0,C 180,E1 -10032.236,E2 -10032.236} C_VEL
LIN {X 0,Y 418.237,Z 396.369,A -85,B 0,C 180,E1 -10035.109,E2 -10035.109} C_VEL
LIN {X 0,Y 418.226,Z 396.393,A -85,B 0,C 180,E1 -10037.765,E2 -10037.765} C_VEL
LIN {X 0,Y 418.238,Z 396.389,A -85,B 0,C 180,E1 -10041.556,E2 -10041.556} C_VEL
LIN {X 0,Y 418.253,Z 396.385,A -85,B 0,C 180,E1 -10045.158,E2 -10045.158} C_VEL
LIN {X 0,Y 418.247,Z 396.38,A -85,B 0,C 180,E1 -10047.472,E2 -10047.472} C_VEL
LIN {X 0,Y 418.263,Z 396.376,A -85,B 0,C 180,E1 -10050.898,E2 -10050.898} C_VEL
LIN {X 0,Y 418.229,Z 396.388,A -85,B 0,C 180,E1 -10054.093,E2 -10054.093} C_VEL
LIN {X 0,Y 418.231,Z 396.378,A -85,B 0,C 180,E1 -10057.263,E2 -10057.263} C_VEL
LIN {X 0,Y 418.287,Z 396.376,A -85,B 0,C 180,E1 -10060.364,E2 -10060.364} C_VEL
LIN {X 0,Y 418.283,Z 396.372,A -85,B 0,C 180,E1 -10063.403,E2 -10063.403} C_VEL
LIN {X 0,Y 418.35,Z 396.368,A -85,B 0,C 180,E1 -10067,E2 -10067} C_VEL
LIN {X 0,Y 418.326,Z 396.372,A -85,B 0,C 180,E1 -10070.328,E2 -10070.328} C_VEL
LIN {X 0,Y 418.445,Z 396.359,A -85,B 0,C 180,E1 -10073.248,E2 -10073.248} C_VEL
LIN {X 0,Y 418.316,Z 396.363,A -85,B 0,C 180,E1 -10075.181,E2 -10075.181} C_VEL
LIN {X 0,Y 418.536,Z 396.35,A -85,B 0,C 180,E1 -10078.075,E2 -10078.075} C_VEL
LIN {X 0,Y 418.41,Z 396.358,A -85,B 0,C 180,E1 -10080.962,E2 -10080.962} C_VEL
LIN {X 0,Y 418.472,Z 396.339,A -85,B 0,C 180,E1 -10082.888,E2 -10082.888} C_VEL
LIN {X 0,Y 418.486,Z 396.359,A -85,B 0,C 180,E1 -10085.783,E2 -10085.783} C_VEL
LIN {X 0,Y 418.37,Z 396.358,A -85,B 0,C 180,E1 -10088.696,E2 -10088.696} C_VEL
LIN {X 0,Y 418.357,Z 396.369,A -85,B 0,C 180,E1 -10092.614,E2 -10092.614} C_VEL
LIN {X 0,Y 418.282,Z 396.365,A -85,B 0,C 180,E1 -10096.597,E2 -10096.597} C_VEL
LIN {X 0,Y 418.239,Z 396.39,A -85,B 0,C 180,E1 -10099.776,E2 -10099.776} C_VEL
LIN {X 0,Y 418.229,Z 396.373,A -85,B 0,C 180,E1 -10102.737,E2 -10102.737} C_VEL
LIN {X 0,Y 418.213,Z 396.394,A -85,B 0,C 180,E1 -10105.908,E2 -10105.908} C_VEL
LIN {X 0,Y 418.259,Z 396.371,A -85,B 0,C 180,E1 -10109.162,E2 -10109.162} C_VEL
LIN {X 0,Y 418.254,Z 396.381,A -85,B 0,C 180,E1 -10112.842,E2 -10112.842} C_VEL
LIN {X 0,Y 418.241,Z 396.388,A -85,B 0,C 180,E1 -10116.236,E2 -10116.236} C_VEL
LIN {X 0,Y 418.195,Z 396.372,A -85,B 0,C 180,E1 -10119.688,E2 -10119.688} C_VEL
LIN {X 0,Y 418.207,Z 396.362,A -85,B 0,C 180,E1 -10122.317,E2 -10122.317} C_VEL
LIN {X 0,Y 418.236,Z 396.385,A -85,B 0,C 180,E1 -10125.108,E2 -10125.108} C_VEL
LIN {X 0,Y 418.218,Z 396.37,A -85,B 0,C 180,E1 -10127.764,E2 -10127.764} C_VEL
LIN {X 0,Y 418.228,Z 396.387,A -85,B 0,C 180,E1 -10131.555,E2 -10131.555} C_VEL
LIN {X 0,Y 418.249,Z 396.387,A -85,B 0,C 180,E1 -10135.158,E2 -10135.158} C_VEL
LIN {X 0,Y 418.279,Z 396.611,A -85,B 0,C 180,E1 -10137.599,E2 -10137.599} C_VEL
LIN {X 0,Y 422.674,Z 415.793,A -85,B 0,C 180,E1 -10140.898,E2 -10140.898} C_VEL
LIN {X 0,Y 423.312,Z 420.327,A -85,B 0,C 180,E1 -10141.634,E2 -10141.634} C_VEL
LIN {X 0,Y 421.828,Z 441.673,A -85,B 0,C 180,E1 -10144.858,E2 -10144.858} C_VEL
LIN {X 0,Y 420.47,Z 463.83,A -85,B 0,C 180,E1 -10148.167,E2 -10148.167} C_VEL
LIN {X 0,Y 419.63,Z 481.482,A -85,B 0,C 180,E1 -10150.748,E2 -10150.748} C_VEL
LIN {X 0,Y 420.326,Z 489.586,A -85,B 0,C 180,E1 -10151.114,E2 -10151.114} C_VEL
LIN {X 0,Y 423.296,Z 517.217,A -85,B 0,C 180,E1 -10151.734,E2 -10151.734} C_VEL
LIN {X 0,Y 422.342,Z 607.415,A -85,B 0,C 180,E1 -10153.287,E2 -10153.287} C_VEL
LIN {X 0,Y 421.884,Z 620.405,A -85,B 0,C 180,E1 -10153.704,E2 -10153.704} C_VEL
LIN {X 0,Y 421.35,Z 633.48,A -85,B 0,C 180,E1 -10154.335,E2 -10154.335} C_VEL
LIN {X 0,Y 420.684,Z 645.251,A -85,B 0,C 180,E1 -10155.116,E2 -10155.116} C_VEL
LIN {X 0,Y 420.021,Z 656.165,A -85,B 0,C 180,E1 -10156.046,E2 -10156.046} C_VEL
LIN {X 0,Y 419.365,Z 666.693,A -85,B 0,C 180,E1 -10157.17,E2 -10157.17} C_VEL
LIN {X 0,Y 418.695,Z 675.789,A -85,B 0,C 180,E1 -10158.379,E2 -10158.379} C_VEL
LIN {X 0,Y 418.089,Z 684.625,A -85,B 0,C 180,E1 -10159.834,E2 -10159.834} C_VEL
LIN {X 0,Y 417.691,Z 691.703,A -85,B 0,C 180,E1 -10161.29,E2 -10161.29} C_VEL
LIN {X 0,Y 417.368,Z 697.322,A -85,B 0,C 180,E1 -10162.744,E2 -10162.744} C_VEL
LIN {X 0,Y 417.205,Z 701.722,A -85,B 0,C 180,E1 -10164.199,E2 -10164.199} C_VEL
LIN {X 0,Y 417.199,Z 704.038,A -85,B 0,C 180,E1 -10165.168,E2 -10165.168} C_VEL
LIN {X 0,Y 417.087,Z 705.923,A -85,B 0,C 180,E1 -10166.135,E2 -10166.135} C_VEL
LIN {X 0,Y 417.111,Z 707.346,A -85,B 0,C 180,E1 -10167.102,E2 -10167.102} C_VEL
LIN {X 0,Y 417.111,Z 708.349,A -85,B 0,C 180,E1 -10168.069,E2 -10168.069} C_VEL
LIN {X 0,Y 417.062,Z 709.181,A -85,B 0,C 180,E1 -10170,E2 -10170} C_VEL
LIN {X 0,Y 417.087,Z 708.961,A -85,B 0,C 180,E1 -10170.965,E2 -10170.965} C_VEL
LIN {X 0,Y 417.115,Z 708.347,A -85,B 0,C 180,E1 -10171.931,E2 -10171.931} C_VEL
LIN {X 0,Y 417.118,Z 707.343,A -85,B 0,C 180,E1 -10172.897,E2 -10172.897} C_VEL
LIN {X 0,Y 417.097,Z 705.917,A -85,B 0,C 180,E1 -10173.865,E2 -10173.865} C_VEL
LIN {X 0,Y 417.24,Z 702.951,A -85,B 0,C 180,E1 -10175.316,E2 -10175.316} C_VEL
LIN {X 0,Y 417.32,Z 698.919,A -85,B 0,C 180,E1 -10176.77,E2 -10176.77} C_VEL
LIN {X 0,Y 417.639,Z 692.697,A -85,B 0,C 180,E1 -10178.467,E2 -10178.467} C_VEL
LIN {X 0,Y 418.019,Z 685.903,A -85,B 0,C 180,E1 -10179.923,E2 -10179.923} C_VEL
LIN {X 0,Y 418.468,Z 678.945,A -85,B 0,C 180,E1 -10181.136,E2 -10181.136} C_VEL
LIN {X 0,Y 419.082,Z 670.529,A -85,B 0,C 180,E1 -10182.346,E2 -10182.346} C_VEL
LIN {X 0,Y 419.786,Z 660.102,A -85,B 0,C 180,E1 -10183.555,E2 -10183.555} C_VEL
LIN {X 0,Y 420.413,Z 649.757,A -85,B 0,C 180,E1 -10184.522,E2 -10184.522} C_VEL
LIN {X 0,Y 421.083,Z 638.338,A -85,B 0,C 180,E1 -10185.364,E2 -10185.364} C_VEL
LIN {X 0,Y 421.696,Z 626.46,A -85,B 0,C 180,E1 -10186.023,E2 -10186.023} C_VEL
LIN {X 0,Y 422.141,Z 613.605,A -85,B 0,C 180,E1 -10186.534,E2 -10186.534} C_VEL
LIN {X 0,Y 422.421,Z 601.509,A -85,B 0,C 180,E1 -10186.834,E2 -10186.834} C_VEL
LIN {X 0,Y 422.928,Z 564.39,A -85,B 0,C 180,E1 -10187.488,E2 -10187.488} C_VEL
LIN {X 0,Y 423.829,Z 515.451,A -85,B 0,C 180,E1 -10188.568,E2 -10188.568} C_VEL
LIN {X 0,Y 421.503,Z 488.756,A -85,B 0,C 180,E1 -10189.352,E2 -10189.352} C_VEL
LIN {X 0,Y 419.632,Z 475.121,A -85,B 0,C 180,E1 -10189.843,E2 -10189.843} C_VEL
LIN {X 0,Y 420.976,Z 452.363,A -85,B 0,C 180,E1 -10193.335,E2 -10193.335} C_VEL
LIN {X 0,Y 422.705,Z 430.006,A -85,B 0,C 180,E1 -10196.941,E2 -10196.941} C_VEL
LIN {X 0,Y 423.622,Z 420.991,A -85,B 0,C 180,E1 -10198.444,E2 -10198.444} C_VEL
LIN {X 0,Y 422.845,Z 414.73,A -85,B 0,C 180,E1 -10199.635,E2 -10199.635} C_VEL
LIN {X 0,Y 420.354,Z 404.254,A -85,B 0,C 180,E1 -10201.851,E2 -10201.851} C_VEL
LIN {X 0,Y 418.245,Z 396.494,A -85,B 0,C 180,E1 -10203.714,E2 -10203.714} C_VEL
LIN {X 0,Y 418.232,Z 396.389,A -85,B 0,C 180,E1 -10207.225,E2 -10207.225} C_VEL
LIN {X 0,Y 418.206,Z 396.39,A -85,B 0,C 180,E1 -10210.867,E2 -10210.867} C_VEL
LIN {X 0,Y 418.202,Z 396.392,A -85,B 0,C 180,E1 -10213.728,E2 -10213.728} C_VEL
LIN {X 0,Y 418.2,Z 396.39,A -85,B 0,C 180,E1 -10216.447,E2 -10216.447} C_VEL
LIN {X 0,Y 418.207,Z 396.391,A -85,B 0,C 180,E1 -10219.133,E2 -10219.133} C_VEL
LIN {X 0,Y 418.236,Z 396.387,A -85,B 0,C 180,E1 -10222.775,E2 -10222.775} C_VEL
LIN {X 0,Y 418.249,Z 396.386,A -85,B 0,C 180,E1 -10226.323,E2 -10226.323} C_VEL
LIN {X 0,Y 418.244,Z 396.388,A -85,B 0,C 180,E1 -10229.728,E2 -10229.728} C_VEL
LIN {X 0,Y 418.245,Z 396.386,A -85,B 0,C 180,E1 -10233.019,E2 -10233.019} C_VEL
LIN {X 0,Y 418.286,Z 396.383,A -85,B 0,C 180,E1 -10236.219,E2 -10236.219} C_VEL
LIN {X 0,Y 418.252,Z 396.387,A -85,B 0,C 180,E1 -10239.337,E2 -10239.337} C_VEL
LIN {X 0,Y 418.343,Z 396.618,A -85,B 0,C 180,E1 -10240.461,E2 -10240.461} C_VEL
LIN {X 0,Y 418.671,Z 397.869,A -85,B 0,C 180,E1 -10240.633,E2 -10240.633} C_VEL
LIN {X 0,Y 424.911,Z 411.392,A -85,B 0,C 180,E1 -10241.442,E2 -10241.442} C_VEL
LIN {X 0,Y 425.499,Z 413.049,A -85,B 0,C 180,E1 -10241.523,E2 -10241.523} C_VEL
LIN {X 0,Y 423.889,Z 479.029,A -85,B 0,C 180,E1 -10243.04,E2 -10243.04} C_VEL
LIN {X 0,Y 423.798,Z 493.285,A -85,B 0,C 180,E1 -10243.501,E2 -10243.501} C_VEL
LIN {X 0,Y 423.576,Z 505.513,A -85,B 0,C 180,E1 -10244.093,E2 -10244.093} C_VEL
LIN {X 0,Y 423.152,Z 517.633,A -85,B 0,C 180,E1 -10244.875,E2 -10244.875} C_VEL
LIN {X 0,Y 422.615,Z 528.787,A -85,B 0,C 180,E1 -10245.801,E2 -10245.801} C_VEL
LIN {X 0,Y 422.068,Z 538.092,A -85,B 0,C 180,E1 -10246.764,E2 -10246.764} C_VEL
LIN {X 0,Y 421.429,Z 547.565,A -85,B 0,C 180,E1 -10247.968,E2 -10247.968} C_VEL
LIN {X 0,Y 420.836,Z 555.3,A -85,B 0,C 180,E1 -10249.171,E2 -10249.171} C_VEL
LIN {X 0,Y 420.307,Z 562.705,A -85,B 0,C 180,E1 -10250.592,E2 -10250.592} C_VEL
LIN {X 0,Y 419.807,Z 567.912,A -85,B 0,C 180,E1 -10251.819,E2 -10251.819} C_VEL
LIN {X 0,Y 419.319,Z 572.772,A -85,B 0,C 180,E1 -10253.262,E2 -10253.262} C_VEL
LIN {X 0,Y 419.005,Z 576.441,A -85,B 0,C 180,E1 -10254.707,E2 -10254.707} C_VEL
LIN {X 0,Y 418.796,Z 579.038,A -85,B 0,C 180,E1 -10256.151,E2 -10256.151} C_VEL
LIN {X 0,Y 418.607,Z 580.212,A -85,B 0,C 180,E1 -10257.113,E2 -10257.113} C_VEL
LIN {X 0,Y 418.492,Z 580.971,A -85,B 0,C 180,E1 -10258.075,E2 -10258.075} C_VEL
LIN {X 0,Y 418.343,Z 581.316,A -85,B 0,C 180,E1 -10259.037,E2 -10259.037} C_VEL
LIN {X 0,Y 418.273,Z 581.199,A -85,B 0,C 180,E1 -10260,E2 -10260} C_VEL
LIN {X 0,Y 418.287,Z 580.671,A -85,B 0,C 180,E1 -10260.963,E2 -10260.963} C_VEL
LIN {X 0,Y 418.209,Z 579.759,A -85,B 0,C 180,E1 -10261.926,E2 -10261.926} C_VEL
LIN {X 0,Y 418.338,Z 578.36,A -85,B 0,C 180,E1 -10262.889,E2 -10262.889} C_VEL
LIN {X 0,Y 418.317,Z 575.491,A -85,B 0,C 180,E1 -10264.336,E2 -10264.336} C_VEL
LIN {X 0,Y 418.565,Z 571.534,A -85,B 0,C 180,E1 -10265.782,E2 -10265.782} C_VEL
LIN {X 0,Y 418.884,Z 566.403,A -85,B 0,C 180,E1 -10267.229,E2 -10267.229} C_VEL
LIN {X 0,Y 419.167,Z 558.763,A -85,B 0,C 180,E1 -10268.922,E2 -10268.922} C_VEL
LIN {X 0,Y 419.591,Z 550.392,A -85,B 0,C 180,E1 -10270.373,E2 -10270.373} C_VEL
LIN {X 0,Y 419.927,Z 541.856,A -85,B 0,C 180,E1 -10271.586,E2 -10271.586} C_VEL
LIN {X 0,Y 420.39,Z 531.39,A -85,B 0,C 180,E1 -10272.798,E2 -10272.798} C_VEL
LIN {X 0,Y 420.92,Z 519.862,A -85,B 0,C 180,E1 -10273.861,E2 -10273.861} C_VEL
LIN {X 0,Y 421.218,Z 507.915,A -85,B 0,C 180,E1 -10274.74,E2 -10274.74} C_VEL
LIN {X 0,Y 421.545,Z 494.671,A -85,B 0,C 180,E1 -10275.471,E2 -10275.471} C_VEL
LIN {X 0,Y 421.801,Z 481.597,A -85,B 0,C 180,E1 -10275.988,E2 -10275.988} C_VEL
LIN {X 0,Y 421.809,Z 466.388,A -85,B 0,C 180,E1 -10276.361,E2 -10276.361} C_VEL
LIN {X 0,Y 422.591,Z 409.721,A -85,B 0,C 180,E1 -10277.515,E2 -10277.515} C_VEL
LIN {X 0,Y 418.492,Z 397.372,A -85,B 0,C 180,E1 -10277.94,E2 -10277.94} C_VEL
LIN {X 0,Y 418.309,Z 396.45,A -85,B 0,C 180,E1 -10278.141,E2 -10278.141} C_VEL
LIN {X 0,Y 418.253,Z 396.388,A -85,B 0,C 180,E1 -10280.663,E2 -10280.663} C_VEL
LIN {X 0,Y 418.289,Z 396.379,A -85,B 0,C 180,E1 -10283.781,E2 -10283.781} C_VEL
LIN {X 0,Y 418.23,Z 396.384,A -85,B 0,C 180,E1 -10287.048,E2 -10287.048} C_VEL
LIN {X 0,Y 418.245,Z 396.381,A -85,B 0,C 180,E1 -10290.272,E2 -10290.272} C_VEL
LIN {X 0,Y 418.249,Z 396.374,A -85,B 0,C 180,E1 -10293.677,E2 -10293.677} C_VEL
LIN {X 0,Y 418.242,Z 396.382,A -85,B 0,C 180,E1 -10297.224,E2 -10297.224} C_VEL
LIN {X 0,Y 418.246,Z 396.384,A -85,B 0,C 180,E1 -10299.683,E2 -10299.683} C_VEL
LIN {X 0,Y 418.225,Z 396.384,A -85,B 0,C 180,E1 -10302.32,E2 -10302.32} C_VEL
LIN {X 0,Y 418.237,Z 396.383,A -85,B 0,C 180,E1 -10305.109,E2 -10305.109} C_VEL
LIN {X 0,Y 418.236,Z 396.384,A -85,B 0,C 180,E1 -10307.766,E2 -10307.766} C_VEL
LIN {X 0,Y 418.24,Z 396.371,A -85,B 0,C 180,E1 -10311.557,E2 -10311.557} C_VEL
LIN {X 0,Y 418.261,Z 396.374,A -85,B 0,C 180,E1 -10315.159,E2 -10315.159} C_VEL
LIN {X 0,Y 418.292,Z 396.596,A -85,B 0,C 180,E1 -10317.797,E2 -10317.797} C_VEL
LIN {X 0,Y 422.376,Z 412.736,A -85,B 0,C 180,E1 -10320.46,E2 -10320.46} C_VEL
LIN {X 0,Y 424.052,Z 420.753,A -85,B 0,C 180,E1 -10321.742,E2 -10321.742} C_VEL
LIN {X 0,Y 423.039,Z 441.342,A -85,B 0,C 180,E1 -10324.673,E2 -10324.673} C_VEL
LIN {X 0,Y 422.01,Z 461.275,A -85,B 0,C 180,E1 -10327.478,E2 -10327.478} C_VEL
LIN {X 0,Y 421.15,Z 481.836,A -85,B 0,C 180,E1 -10330.25,E2 -10330.25} C_VEL
LIN {X 0,Y 421.02,Z 487.992,A -85,B 0,C 180,E1 -10331.026,E2 -10331.026} C_VEL
LIN {X 0,Y 423.887,Z 507.791,A -85,B 0,C 180,E1 -10331.517,E2 -10331.517} C_VEL
LIN {X 0,Y 423.045,Z 583.304,A -85,B 0,C 180,E1 -10332.805,E2 -10332.805} C_VEL
LIN {X 0,Y 422.398,Z 589.154,A -85,B 0,C 180,E1 -10332.88,E2 -10332.88} C_VEL
LIN {X 0,Y 419.54,Z 598.647,A -85,B 0,C 180,E1 -10332.95,E2 -10332.95} C_VEL
LIN {X 0,Y 416.507,Z 608.027,A -85,B 0,C 180,E1 -10333.099,E2 -10333.099} C_VEL
LIN {X 0,Y 415.559,Z 613.697,A -85,B 0,C 180,E1 -10333.287,E2 -10333.287} C_VEL
LIN {X 0,Y 414.964,Z 626.05,A -85,B 0,C 180,E1 -10333.899,E2 -10333.899} C_VEL
LIN {X 0,Y 414.215,Z 638.749,A -85,B 0,C 180,E1 -10334.753,E2 -10334.753} C_VEL
LIN {X 0,Y 413.495,Z 649.64,A -85,B 0,C 180,E1 -10335.708,E2 -10335.708} C_VEL
LIN {X 0,Y 412.782,Z 659.971,A -85,B 0,C 180,E1 -10336.837,E2 -10336.837} C_VEL
LIN {X 0,Y 412.088,Z 668.255,A -85,B 0,C 180,E1 -10337.941,E2 -10337.941} C_VEL
LIN {X 0,Y 411.394,Z 677.243,A -85,B 0,C 180,E1 -10339.418,E2 -10339.418} C_VEL
LIN {X 0,Y 410.862,Z 684.459,A -85,B 0,C 180,E1 -10340.896,E2 -10340.896} C_VEL
LIN {X 0,Y 410.401,Z 691.083,A -85,B 0,C 180,E1 -10342.621,E2 -10342.621} C_VEL
LIN {X 0,Y 410.188,Z 695.434,A -85,B 0,C 180,E1 -10344.1,E2 -10344.1} C_VEL
LIN {X 0,Y 410.119,Z 697.725,A -85,B 0,C 180,E1 -10345.085,E2 -10345.085} C_VEL
LIN {X 0,Y 409.96,Z 699.594,A -85,B 0,C 180,E1 -10346.068,E2 -10346.068} C_VEL
LIN {X 0,Y 409.938,Z 701.022,A -85,B 0,C 180,E1 -10347.052,E2 -10347.052} C_VEL
LIN {X 0,Y 409.968,Z 702.023,A -85,B 0,C 180,E1 -10348.035,E2 -10348.035} C_VEL
LIN {X 0,Y 409.906,Z 702.878,A -85,B 0,C 180,E1 -10350,E2 -10350} C_VEL
LIN {X 0,Y 409.919,Z 702.686,A -85,B 0,C 180,E1 -10350.983,E2 -10350.983} C_VEL
LIN {X 0,Y 409.968,Z 702.098,A -85,B 0,C 180,E1 -10351.965,E2 -10351.965} C_VEL
LIN {X 0,Y 409.959,Z 699.757,A -85,B 0,C 180,E1 -10353.932,E2 -10353.932} C_VEL
LIN {X 0,Y 410.143,Z 696.875,A -85,B 0,C 180,E1 -10355.408,E2 -10355.408} C_VEL
LIN {X 0,Y 410.264,Z 692.961,A -85,B 0,C 180,E1 -10356.887,E2 -10356.887} C_VEL
LIN {X 0,Y 410.587,Z 687.89,A -85,B 0,C 180,E1 -10358.366,E2 -10358.366} C_VEL
LIN {X 0,Y 411.064,Z 681.499,A -85,B 0,C 180,E1 -10359.844,E2 -10359.844} C_VEL
LIN {X 0,Y 411.65,Z 673.561,A -85,B 0,C 180,E1 -10361.323,E2 -10361.323} C_VEL
LIN {X 0,Y 412.372,Z 665.453,A -85,B 0,C 180,E1 -10362.551,E2 -10362.551} C_VEL
LIN {X 0,Y 413.18,Z 655.494,A -85,B 0,C 180,E1 -10363.777,E2 -10363.777} C_VEL
LIN {X 0,Y 413.746,Z 645.676,A -85,B 0,C 180,E1 -10364.762,E2 -10364.762} C_VEL
LIN {X 0,Y 414.486,Z 635.043,A -85,B 0,C 180,E1 -10365.615,E2 -10365.615} C_VEL
LIN {X 0,Y 415.167,Z 623.402,A -85,B 0,C 180,E1 -10366.346,E2 -10366.346} C_VEL
LIN {X 0,Y 415.741,Z 610.741,A -85,B 0,C 180,E1 -10366.923,E2 -10366.923} C_VEL
LIN {X 0,Y 416.138,Z 597.494,A -85,B 0,C 180,E1 -10367.317,E2 -10367.317} C_VEL
LIN {X 0,Y 417.109,Z 508.132,A -85,B 0,C 180,E1 -10368.884,E2 -10368.884} C_VEL
LIN {X 0,Y 414.204,Z 487.814,A -85,B 0,C 180,E1 -10369.405,E2 -10369.405} C_VEL
LIN {X 0,Y 414.878,Z 469.192,A -85,B 0,C 180,E1 -10371.881,E2 -10371.881} C_VEL
LIN {X 0,Y 416.209,Z 443.526,A -85,B 0,C 180,E1 -10375.505,E2 -10375.505} C_VEL
LIN {X 0,Y 417.35,Z 423.011,A -85,B 0,C 180,E1 -10378.464,E2 -10378.464} C_VEL
LIN {X 0,Y 414.525,Z 409.936,A -85,B 0,C 180,E1 -10380.573,E2 -10380.573} C_VEL
LIN {X 0,Y 411.245,Z 397.474,A -85,B 0,C 180,E1 -10382.679,E2 -10382.679} C_VEL
LIN {X 0,Y 411.197,Z 397.267,A -85,B 0,C 180,E1 -10385.529,E2 -10385.529} C_VEL
LIN {X 0,Y 411.18,Z 397.262,A -85,B 0,C 180,E1 -10389.229,E2 -10389.229} C_VEL
LIN {X 0,Y 411.169,Z 397.267,A -85,B 0,C 180,E1 -10392.693,E2 -10392.693} C_VEL
LIN {X 0,Y 411.167,Z 397.257,A -85,B 0,C 180,E1 -10395.882,E2 -10395.882} C_VEL
LIN {X 0,Y 411.151,Z 397.268,A -85,B 0,C 180,E1 -10398.774,E2 -10398.774} C_VEL
LIN {X 0,Y 411.186,Z 397.26,A -85,B 0,C 180,E1 -10402.025,E2 -10402.025} C_VEL
LIN {X 0,Y 411.205,Z 397.263,A -85,B 0,C 180,E1 -10405.123,E2 -10405.123} C_VEL
LIN {X 0,Y 411.167,Z 397.27,A -85,B 0,C 180,E1 -10408.003,E2 -10408.003} C_VEL
LIN {X 0,Y 411.175,Z 397.259,A -85,B 0,C 180,E1 -10411.407,E2 -10411.407} C_VEL
LIN {X 0,Y 411.215,Z 397.259,A -85,B 0,C 180,E1 -10414.934,E2 -10414.934} C_VEL
LIN {X 0,Y 411.207,Z 397.262,A -85,B 0,C 180,E1 -10417.913,E2 -10417.913} C_VEL
LIN {X 0,Y 411.219,Z 397.257,A -85,B 0,C 180,E1 -10421.051,E2 -10421.051} C_VEL
LIN {X 0,Y 411.215,Z 397.262,A -85,B 0,C 180,E1 -10424.13,E2 -10424.13} C_VEL
LIN {X 0,Y 411.306,Z 397.246,A -85,B 0,C 180,E1 -10427.166,E2 -10427.166} C_VEL
LIN {X 0,Y 411.28,Z 397.251,A -85,B 0,C 180,E1 -10430.161,E2 -10430.161} C_VEL
LIN {X 0,Y 411.394,Z 397.237,A -85,B 0,C 180,E1 -10433.132,E2 -10433.132} C_VEL
LIN {X 0,Y 411.288,Z 397.238,A -85,B 0,C 180,E1 -10435.099,E2 -10435.099} C_VEL
LIN {X 0,Y 411.505,Z 397.227,A -85,B 0,C 180,E1 -10438.042,E2 -10438.042} C_VEL
LIN {X 0,Y 411.38,Z 397.234,A -85,B 0,C 180,E1 -10440.979,E2 -10440.979} C_VEL
LIN {X 0,Y 411.431,Z 397.216,A -85,B 0,C 180,E1 -10442.937,E2 -10442.937} C_VEL
LIN {X 0,Y 411.431,Z 397.238,A -85,B 0,C 180,E1 -10445.883,E2 -10445.883} C_VEL
LIN {X 0,Y 411.31,Z 397.237,A -85,B 0,C 180,E1 -10448.846,E2 -10448.846} C_VEL
LIN {X 0,Y 411.277,Z 397.251,A -85,B 0,C 180,E1 -10451.833,E2 -10451.833} C_VEL
LIN {X 0,Y 411.211,Z 397.255,A -85,B 0,C 180,E1 -10454.854,E2 -10454.854} C_VEL
LIN {X 0,Y 411.169,Z 397.259,A -85,B 0,C 180,E1 -10457.919,E2 -10457.919} C_VEL
LIN {X 0,Y 411.183,Z 397.262,A -85,B 0,C 180,E1 -10461.035,E2 -10461.035} C_VEL
LIN {X 0,Y 411.193,Z 397.259,A -85,B 0,C 180,E1 -10464.218,E2 -10464.218} C_VEL
LIN {X 0,Y 411.146,Z 397.27,A -85,B 0,C 180,E1 -10467.486,E2 -10467.486} C_VEL
LIN {X 0,Y 411.198,Z 397.253,A -85,B 0,C 180,E1 -10469.713,E2 -10469.713} C_VEL
LIN {X 0,Y 411.207,Z 397.26,A -85,B 0,C 180,E1 -10473.156,E2 -10473.156} C_VEL
LIN {X 0,Y 411.19,Z 397.264,A -85,B 0,C 180,E1 -10476.551,E2 -10476.551} C_VEL
LIN {X 0,Y 411.165,Z 397.246,A -85,B 0,C 180,E1 -10479.719,E2 -10479.719} C_VEL
LIN {X 0,Y 411.162,Z 397.252,A -85,B 0,C 180,E1 -10483.135,E2 -10483.135} C_VEL
LIN {X 0,Y 411.164,Z 397.269,A -85,B 0,C 180,E1 -10485.882,E2 -10485.882} C_VEL
LIN {X 0,Y 411.157,Z 397.241,A -85,B 0,C 180,E1 -10489.492,E2 -10489.492} C_VEL
LIN {X 0,Y 411.179,Z 397.27,A -85,B 0,C 180,E1 -10492.024,E2 -10492.024} C_VEL
LIN {X 0,Y 411.201,Z 397.265,A -85,B 0,C 180,E1 -10495.124,E2 -10495.124} C_VEL
LIN {X 0,Y 411.243,Z 397.496,A -85,B 0,C 180,E1 -10497.346,E2 -10497.346} C_VEL
LIN {X 0,Y 415.831,Z 417.605,A -85,B 0,C 180,E1 -10500.856,E2 -10500.856} C_VEL
LIN {X 0,Y 416.364,Z 421.58,A -85,B 0,C 180,E1 -10501.511,E2 -10501.511} C_VEL
LIN {X 0,Y 414.868,Z 442.188,A -85,B 0,C 180,E1 -10504.675,E2 -10504.675} C_VEL
LIN {X 0,Y 413.546,Z 462.622,A -85,B 0,C 180,E1 -10507.782,E2 -10507.782} C_VEL
LIN {X 0,Y 412.669,Z 479.423,A -85,B 0,C 180,E1 -10510.299,E2 -10510.299} C_VEL
LIN {X 0,Y 413.487,Z 489.281,A -85,B 0,C 180,E1 -10510.782,E2 -10510.782} C_VEL
LIN {X 0,Y 416.568,Z 517.515,A -85,B 0,C 180,E1 -10511.432,E2 -10511.432} C_VEL
LIN {X 0,Y 415.569,Z 607.445,A -85,B 0,C 180,E1 -10513.007,E2 -10513.007} C_VEL
LIN {X 0,Y 415.053,Z 621.152,A -85,B 0,C 180,E1 -10513.46,E2 -10513.46} C_VEL
LIN {X 0,Y 414.522,Z 633.458,A -85,B 0,C 180,E1 -10514.07,E2 -10514.07} C_VEL
LIN {X 0,Y 413.837,Z 645.219,A -85,B 0,C 180,E1 -10514.864,E2 -10514.864} C_VEL
LIN {X 0,Y 413.115,Z 656.243,A -85,B 0,C 180,E1 -10515.819,E2 -10515.819} C_VEL
LIN {X 0,Y 412.442,Z 666.65,A -85,B 0,C 180,E1 -10516.951,E2 -10516.951} C_VEL
LIN {X 0,Y 411.73,Z 675.743,A -85,B 0,C 180,E1 -10518.18,E2 -10518.18} C_VEL
LIN {X 0,Y 411.089,Z 684.577,A -85,B 0,C 180,E1 -10519.659,E2 -10519.659} C_VEL
LIN {X 0,Y 410.665,Z 691.653,A -85,B 0,C 180,E1 -10521.14,E2 -10521.14} C_VEL
LIN {X 0,Y 410.297,Z 697.271,A -85,B 0,C 180,E1 -10522.619,E2 -10522.619} C_VEL
LIN {X 0,Y 410.12,Z 701.67,A -85,B 0,C 180,E1 -10524.098,E2 -10524.098} C_VEL
LIN {X 0,Y 410.132,Z 703.985,A -85,B 0,C 180,E1 -10525.085,E2 -10525.085} C_VEL
LIN {X 0,Y 410.003,Z 705.87,A -85,B 0,C 180,E1 -10526.068,E2 -10526.068} C_VEL
LIN {X 0,Y 410.007,Z 707.292,A -85,B 0,C 180,E1 -10527.052,E2 -10527.052} C_VEL
LIN {X 0,Y 410.038,Z 708.296,A -85,B 0,C 180,E1 -10528.035,E2 -10528.035} C_VEL
LIN {X 0,Y 409.982,Z 709.128,A -85,B 0,C 180,E1 -10530,E2 -10530} C_VEL
LIN {X 0,Y 410.007,Z 708.907,A -85,B 0,C 180,E1 -10530.982,E2 -10530.982} C_VEL
LIN {X 0,Y 410.042,Z 708.293,A -85,B 0,C 180,E1 -10531.964,E2 -10531.964} C_VEL
LIN {X 0,Y 410.014,Z 707.289,A -85,B 0,C 180,E1 -10532.947,E2 -10532.947} C_VEL
LIN {X 0,Y 410.013,Z 705.863,A -85,B 0,C 180,E1 -10533.931,E2 -10533.931} C_VEL
LIN {X 0,Y 410.153,Z 702.897,A -85,B 0,C 180,E1 -10535.408,E2 -10535.408} C_VEL
LIN {X 0,Y 410.253,Z 698.866,A -85,B 0,C 180,E1 -10536.887,E2 -10536.887} C_VEL
LIN {X 0,Y 410.583,Z 692.644,A -85,B 0,C 180,E1 -10538.614,E2 -10538.614} C_VEL
LIN {X 0,Y 410.987,Z 685.851,A -85,B 0,C 180,E1 -10540.095,E2 -10540.095} C_VEL
LIN {X 0,Y 411.493,Z 678.894,A -85,B 0,C 180,E1 -10541.327,E2 -10541.327} C_VEL
LIN {X 0,Y 412.116,Z 670.481,A -85,B 0,C 180,E1 -10542.558,E2 -10542.558} C_VEL
LIN {X 0,Y 412.863,Z 660.056,A -85,B 0,C 180,E1 -10543.787,E2 -10543.787} C_VEL
LIN {X 0,Y 413.544,Z 649.715,A -85,B 0,C 180,E1 -10544.769,E2 -10544.769} C_VEL
LIN {X 0,Y 414.221,Z 638.302,A -85,B 0,C 180,E1 -10545.625,E2 -10545.625} C_VEL
LIN {X 0,Y 414.869,Z 626.434,A -85,B 0,C 180,E1 -10546.294,E2 -10546.294} C_VEL
LIN {X 0,Y 415.355,Z 613.597,A -85,B 0,C 180,E1 -10546.812,E2 -10546.812} C_VEL
LIN {X 0,Y 415.641,Z 601.546,A -85,B 0,C 180,E1 -10547.117,E2 -10547.117} C_VEL
LIN {X 0,Y 416.042,Z 573.301,A -85,B 0,C 180,E1 -10547.638,E2 -10547.638} C_VEL
LIN {X 0,Y 417.279,Z 516.414,A -85,B 0,C 180,E1 -10548.918,E2 -10548.918} C_VEL
LIN {X 0,Y 415.163,Z 490.729,A -85,B 0,C 180,E1 -10549.701,E2 -10549.701} C_VEL
LIN {X 0,Y 412.797,Z 473.759,A -85,B 0,C 180,E1 -10550.328,E2 -10550.328} C_VEL
LIN {X 0,Y 414.135,Z 452.149,A -85,B 0,C 180,E1 -10553.725,E2 -10553.725} C_VEL
LIN {X 0,Y 415.802,Z 432.985,A -85,B 0,C 180,E1 -10556.885,E2 -10556.885} C_VEL
LIN {X 0,Y 416.871,Z 422.099,A -85,B 0,C 180,E1 -10558.757,E2 -10558.757} C_VEL
LIN {X 0,Y 415.552,Z 413.954,A -85,B 0,C 180,E1 -10560.397,E2 -10560.397} C_VEL
LIN {X 0,Y 413.02,Z 403.731,A -85,B 0,C 180,E1 -10562.701,E2 -10562.701} C_VEL
LIN {X 0,Y 411.212,Z 397.349,A -85,B 0,C 180,E1 -10564.367,E2 -10564.367} C_VEL
LIN {X 0,Y 411.18,Z 397.269,A -85,B 0,C 180,E1 -10567.975,E2 -10567.975} C_VEL
LIN {X 0,Y 411.146,Z 397.271,A -85,B 0,C 180,E1 -10571.225,E2 -10571.225} C_VEL
LIN {X 0,Y 411.174,Z 397.268,A -85,B 0,C 180,E1 -10574.491,E2 -10574.491} C_VEL
LIN {X 0,Y 411.161,Z 397.268,A -85,B 0,C 180,E1 -10578.192,E2 -10578.192} C_VEL
LIN {X 0,Y 411.193,Z 397.264,A -85,B 0,C 180,E1 -10581.834,E2 -10581.834} C_VEL
LIN {X 0,Y 411.21,Z 397.265,A -85,B 0,C 180,E1 -10585.122,E2 -10585.122} C_VEL
LIN {X 0,Y 411.167,Z 397.269,A -85,B 0,C 180,E1 -10588.003,E2 -10588.003} C_VEL
LIN {X 0,Y 411.196,Z 397.264,A -85,B 0,C 180,E1 -10591.408,E2 -10591.408} C_VEL
LIN {X 0,Y 411.228,Z 397.261,A -85,B 0,C 180,E1 -10594.929,E2 -10594.929} C_VEL
LIN {X 0,Y 411.208,Z 397.265,A -85,B 0,C 180,E1 -10597.914,E2 -10597.914} C_VEL
LIN {X 0,Y 411.232,Z 397.384,A -85,B 0,C 180,E1 -10599.876,E2 -10599.876} C_VEL
LIN {X 0,Y 411.467,Z 398.371,A -85,B 0,C 180,E1 -10600.075,E2 -10600.075} C_VEL
LIN {X 0,Y 417.069,Z 409.919,A -85,B 0,C 180,E1 -10600.848,E2 -10600.848} C_VEL
LIN {X 0,Y 419.001,Z 414.524,A -85,B 0,C 180,E1 -10601.114,E2 -10601.114} C_VEL
LIN {X 0,Y 417.675,Z 461.546,A -85,B 0,C 180,E1 -10602.238,E2 -10602.238} C_VEL
LIN {X 0,Y 417.355,Z 486.474,A -85,B 0,C 180,E1 -10602.861,E2 -10602.861} C_VEL
LIN {X 0,Y 417.226,Z 499.028,A -85,B 0,C 180,E1 -10603.36,E2 -10603.36} C_VEL
LIN {X 0,Y 416.843,Z 511.108,A -85,B 0,C 180,E1 -10604.022,E2 -10604.022} C_VEL
LIN {X 0,Y 416.358,Z 522.901,A -85,B 0,C 180,E1 -10604.883,E2 -10604.883} C_VEL
LIN {X 0,Y 415.631,Z 534.322,A -85,B 0,C 180,E1 -10605.932,E2 -10605.932} C_VEL
LIN {X 0,Y 415.058,Z 543.82,A -85,B 0,C 180,E1 -10607.035,E2 -10607.035} C_VEL
LIN {X 0,Y 414.451,Z 552.439,A -85,B 0,C 180,E1 -10608.259,E2 -10608.259} C_VEL
LIN {X 0,Y 413.819,Z 559.529,A -85,B 0,C 180,E1 -10609.48,E2 -10609.48} C_VEL
LIN {X 0,Y 413.261,Z 566.141,A -85,B 0,C 180,E1 -10610.883,E2 -10610.883} C_VEL
LIN {X 0,Y 412.743,Z 571.024,A -85,B 0,C 180,E1 -10612.171,E2 -10612.171} C_VEL
LIN {X 0,Y 412.366,Z 575.396,A -85,B 0,C 180,E1 -10613.64,E2 -10613.64} C_VEL
LIN {X 0,Y 411.902,Z 578.683,A -85,B 0,C 180,E1 -10615.106,E2 -10615.106} C_VEL
LIN {X 0,Y 411.813,Z 580.238,A -85,B 0,C 180,E1 -10616.086,E2 -10616.086} C_VEL
LIN {X 0,Y 411.614,Z 581.382,A -85,B 0,C 180,E1 -10617.064,E2 -10617.064} C_VEL
LIN {X 0,Y 411.504,Z 582.107,A -85,B 0,C 180,E1 -10618.043,E2 -10618.043} C_VEL
LIN {X 0,Y 411.329,Z 582.401,A -85,B 0,C 180,E1 -10619.021,E2 -10619.021} C_VEL
LIN {X 0,Y 411.252,Z 582.249,A -85,B 0,C 180,E1 -10620,E2 -10620} C_VEL
LIN {X 0,Y 411.263,Z 581.681,A -85,B 0,C 180,E1 -10620.979,E2 -10620.979} C_VEL
LIN {X 0,Y 411.186,Z 580.714,A -85,B 0,C 180,E1 -10621.959,E2 -10621.959} C_VEL
LIN {X 0,Y 411.315,Z 579.261,A -85,B 0,C 180,E1 -10622.938,E2 -10622.938} C_VEL
LIN {X 0,Y 411.297,Z 576.312,A -85,B 0,C 180,E1 -10624.41,E2 -10624.41} C_VEL
LIN {X 0,Y 411.547,Z 572.27,A -85,B 0,C 180,E1 -10625.881,E2 -10625.881} C_VEL
LIN {X 0,Y 411.931,Z 566.077,A -85,B 0,C 180,E1 -10627.598,E2 -10627.598} C_VEL
LIN {X 0,Y 412.186,Z 559.267,A -85,B 0,C 180,E1 -10629.075,E2 -10629.075} C_VEL
LIN {X 0,Y 412.607,Z 550.778,A -85,B 0,C 180,E1 -10630.551,E2 -10630.551} C_VEL
LIN {X 0,Y 412.97,Z 542.113,A -85,B 0,C 180,E1 -10631.784,E2 -10631.784} C_VEL
LIN {X 0,Y 413.463,Z 531.419,A -85,B 0,C 180,E1 -10633.016,E2 -10633.016} C_VEL
LIN {X 0,Y 413.991,Z 520.052,A -85,B 0,C 180,E1 -10634.067,E2 -10634.067} C_VEL
LIN {X 0,Y 414.265,Z 509.303,A -85,B 0,C 180,E1 -10634.868,E2 -10634.868} C_VEL
LIN {X 0,Y 414.63,Z 496.265,A -85,B 0,C 180,E1 -10635.61,E2 -10635.61} C_VEL
LIN {X 0,Y 414.856,Z 483.461,A -85,B 0,C 180,E1 -10636.137,E2 -10636.137} C_VEL
LIN {X 0,Y 414.866,Z 469.044,A -85,B 0,C 180,E1 -10636.516,E2 -10636.516} C_VEL
LIN {X 0,Y 415.654,Z 410.962,A -85,B 0,C 180,E1 -10637.727,E2 -10637.727} C_VEL
LIN {X 0,Y 411.44,Z 398.141,A -85,B 0,C 180,E1 -10638.185,E2 -10638.185} C_VEL
LIN {X 0,Y 411.267,Z 397.345,A -85,B 0,C 180,E1 -10638.365,E2 -10638.365} C_VEL
LIN {X 0,Y 411.199,Z 397.267,A -85,B 0,C 180,E1 -10641.034,E2 -10641.034} C_VEL
LIN {X 0,Y 411.221,Z 397.261,A -85,B 0,C 180,E1 -10644.216,E2 -10644.216} C_VEL
LIN {X 0,Y 411.192,Z 397.257,A -85,B 0,C 180,E1 -10647.483,E2 -10647.483} C_VEL
LIN {X 0,Y 411.191,Z 397.267,A -85,B 0,C 180,E1 -10650.848,E2 -10650.848} C_VEL
LIN {X 0,Y 411.206,Z 397.252,A -85,B 0,C 180,E1 -10654.334,E2 -10654.334} C_VEL
LIN {X 0,Y 411.194,Z 397.258,A -85,B 0,C 180,E1 -10657.974,E2 -10657.974} C_VEL
LIN {X 0,Y 411.162,Z 397.264,A -85,B 0,C 180,E1 -10661.228,E2 -10661.228} C_VEL
LIN {X 0,Y 411.177,Z 397.267,A -85,B 0,C 180,E1 -10664.491,E2 -10664.491} C_VEL
LIN {X 0,Y 411.174,Z 397.264,A -85,B 0,C 180,E1 -10668.194,E2 -10668.194} C_VEL
LIN {X 0,Y 411.185,Z 397.252,A -85,B 0,C 180,E1 -10670.772,E2 -10670.772} C_VEL
LIN {X 0,Y 411.199,Z 397.255,A -85,B 0,C 180,E1 -10674.471,E2 -10674.471} C_VEL
LIN {X 0,Y 411.245,Z 397.449,A -85,B 0,C 180,E1 -10677.413,E2 -10677.413} C_VEL
LIN {X 0,Y 415.436,Z 413.958,A -85,B 0,C 180,E1 -10680.196,E2 -10680.196} C_VEL
LIN {X 0,Y 417.314,Z 423.197,A -85,B 0,C 180,E1 -10681.679,E2 -10681.679} C_VEL
LIN {X 0,Y 416.14,Z 444.616,A -85,B 0,C 180,E1 -10684.758,E2 -10684.758} C_VEL
LIN {X 0,Y 414.982,Z 466.664,A -85,B 0,C 180,E1 -10687.863,E2 -10687.863} C_VEL
LIN {X 0,Y 414.155,Z 487.756,A -85,B 0,C 180,E1 -10690.685,E2 -10690.685} C_VEL
LIN {X 0,Y 417.187,Z 509.829,A -85,B 0,C 180,E1 -10691.246,E2 -10691.246} C_VEL
LIN {X 0,Y 416.081,Z 600.046,A -85,B 0,C 180,E1 -10692.839,E2 -10692.839} C_VEL
LIN {X 0,Y 415.6,Z 613.086,A -85,B 0,C 180,E1 -10693.261,E2 -10693.261} C_VEL
LIN {X 0,Y 415.559,Z 613.697,A -85,B 0,C 180,E1 -10693.287,E2 -10693.287} C_VEL
LIN {X 0,Y 413.996,Z 621.205,A -85,B 0,C 180,E1 -10693.585,E2 -10693.585} C_VEL
LIN {X 0,Y 411.289,Z 628.427,A -85,B 0,C 180,E1 -10693.895,E2 -10693.895} C_VEL
LIN {X 0,Y 408.064,Z 637.027,A -85,B 0,C 180,E1 -10694.377,E2 -10694.377} C_VEL
LIN {X 0,Y 407.145,Z 642.093,A -85,B 0,C 180,E1 -10694.761,E2 -10694.761} C_VEL
LIN {X 0,Y 406.489,Z 652.138,A -85,B 0,C 180,E1 -10695.708,E2 -10695.708} C_VEL
LIN {X 0,Y 405.799,Z 661.034,A -85,B 0,C 180,E1 -10696.734,E2 -10696.734} C_VEL
LIN {X 0,Y 404.978,Z 669.936,A -85,B 0,C 180,E1 -10697.98,E2 -10697.98} C_VEL
LIN {X 0,Y 404.285,Z 678.618,A -85,B 0,C 180,E1 -10699.483,E2 -10699.483} C_VEL
LIN {X 0,Y 403.757,Z 685.592,A -85,B 0,C 180,E1 -10700.987,E2 -10700.987} C_VEL
LIN {X 0,Y 403.334,Z 691.136,A -85,B 0,C 180,E1 -10702.491,E2 -10702.491} C_VEL
LIN {X 0,Y 403.111,Z 695.489,A -85,B 0,C 180,E1 -10703.996,E2 -10703.996} C_VEL
LIN {X 0,Y 403.035,Z 697.779,A -85,B 0,C 180,E1 -10704.998,E2 -10704.998} C_VEL
LIN {X 0,Y 402.883,Z 699.648,A -85,B 0,C 180,E1 -10705.999,E2 -10705.999} C_VEL
LIN {X 0,Y 402.838,Z 701.077,A -85,B 0,C 180,E1 -10707,E2 -10707} C_VEL
LIN {X 0,Y 402.866,Z 702.077,A -85,B 0,C 180,E1 -10708.001,E2 -10708.001} C_VEL
LIN {X 0,Y 402.832,Z 702.932,A -85,B 0,C 180,E1 -10710,E2 -10710} C_VEL
LIN {X 0,Y 402.848,Z 702.74,A -85,B 0,C 180,E1 -10711,E2 -10711} C_VEL
LIN {X 0,Y 402.866,Z 702.151,A -85,B 0,C 180,E1 -10712,E2 -10712} C_VEL
LIN {X 0,Y 402.882,Z 699.81,A -85,B 0,C 180,E1 -10714.001,E2 -10714.001} C_VEL
LIN {X 0,Y 403.066,Z 696.927,A -85,B 0,C 180,E1 -10715.503,E2 -10715.503} C_VEL
LIN {X 0,Y 403.203,Z 693.012,A -85,B 0,C 180,E1 -10717.008,E2 -10717.008} C_VEL
LIN {X 0,Y 403.564,Z 687.94,A -85,B 0,C 180,E1 -10718.513,E2 -10718.513} C_VEL
LIN {X 0,Y 404.036,Z 681.547,A -85,B 0,C 180,E1 -10720.017,E2 -10720.017} C_VEL
LIN {X 0,Y 404.676,Z 673.608,A -85,B 0,C 180,E1 -10721.521,E2 -10721.521} C_VEL
LIN {X 0,Y 405.426,Z 665.497,A -85,B 0,C 180,E1 -10722.769,E2 -10722.769} C_VEL
LIN {X 0,Y 406.256,Z 655.533,A -85,B 0,C 180,E1 -10724.016,E2 -10724.016} C_VEL
LIN {X 0,Y 406.965,Z 644.338,A -85,B 0,C 180,E1 -10725.141,E2 -10725.141} C_VEL
LIN {X 0,Y 407.767,Z 633.378,A -85,B 0,C 180,E1 -10726.008,E2 -10726.008} C_VEL
LIN {X 0,Y 408.477,Z 621.049,A -85,B 0,C 180,E1 -10726.75,E2 -10726.75} C_VEL
LIN {X 0,Y 409.034,Z 609.065,A -85,B 0,C 180,E1 -10727.273,E2 -10727.273} C_VEL
LIN {X 0,Y 409.434,Z 596.114,A -85,B 0,C 180,E1 -10727.642,E2 -10727.642} C_VEL
LIN {X 0,Y 410.423,Z 509.086,A -85,B 0,C 180,E1 -10729.184,E2 -10729.184} C_VEL
LIN {X 0,Y 407.359,Z 487.802,A -85,B 0,C 180,E1 -10729.744,E2 -10729.744} C_VEL
LIN {X 0,Y 408.091,Z 469.047,A -85,B 0,C 180,E1 -10732.264,E2 -10732.264} C_VEL
LIN {X 0,Y 409.523,Z 443.184,A -85,B 0,C 180,E1 -10735.952,E2 -10735.952} C_VEL
LIN {X 0,Y 410.598,Z 424.742,A -85,B 0,C 180,E1 -10738.638,E2 -10738.638} C_VEL
LIN {X 0,Y 407.425,Z 410.588,A -85,B 0,C 180,E1 -10740.966,E2 -10740.966} C_VEL
LIN {X 0,Y 404.192,Z 398.314,A -85,B 0,C 180,E1 -10743.085,E2 -10743.085} C_VEL
LIN {X 0,Y 404.141,Z 398.136,A -85,B 0,C 180,E1 -10746.247,E2 -10746.247} C_VEL
LIN {X 0,Y 404.135,Z 398.146,A -85,B 0,C 180,E1 -10748.76,E2 -10748.76} C_VEL
LIN {X 0,Y 404.108,Z 398.143,A -85,B 0,C 180,E1 -10751.597,E2 -10751.597} C_VEL
LIN {X 0,Y 404.145,Z 398.123,A -85,B 0,C 180,E1 -10754.522,E2 -10754.522} C_VEL
LIN {X 0,Y 404.127,Z 398.146,A -85,B 0,C 180,E1 -10757.294,E2 -10757.294} C_VEL
LIN {X 0,Y 404.135,Z 398.145,A -85,B 0,C 180,E1 -10759.951,E2 -10759.951} C_VEL
LIN {X 0,Y 404.135,Z 398.136,A -85,B 0,C 180,E1 -10763.126,E2 -10763.126} C_VEL
LIN {X 0,Y 404.141,Z 398.133,A -85,B 0,C 180,E1 -10766.187,E2 -10766.187} C_VEL
LIN {X 0,Y 404.147,Z 398.142,A -85,B 0,C 180,E1 -10769.715,E2 -10769.715} C_VEL
LIN {X 0,Y 404.108,Z 398.146,A -85,B 0,C 180,E1 -10773.116,E2 -10773.116} C_VEL
LIN {X 0,Y 404.153,Z 398.129,A -85,B 0,C 180,E1 -10776.424,E2 -10776.424} C_VEL
LIN {X 0,Y 404.195,Z 398.136,A -85,B 0,C 180,E1 -10779.874,E2 -10779.874} C_VEL
LIN {X 0,Y 404.177,Z 398.126,A -85,B 0,C 180,E1 -10783.013,E2 -10783.013} C_VEL
LIN {X 0,Y 404.287,Z 398.12,A -85,B 0,C 180,E1 -10786.939,E2 -10786.939} C_VEL
LIN {X 0,Y 404.247,Z 398.123,A -85,B 0,C 180,E1 -10789.988,E2 -10789.988} C_VEL
LIN {X 0,Y 404.344,Z 398.115,A -85,B 0,C 180,E1 -10793.012,E2 -10793.012} C_VEL
LIN {X 0,Y 404.259,Z 398.113,A -85,B 0,C 180,E1 -10795.013,E2 -10795.013} C_VEL
LIN {X 0,Y 404.474,Z 398.103,A -85,B 0,C 180,E1 -10798.008,E2 -10798.008} C_VEL
LIN {X 0,Y 404.351,Z 398.109,A -85,B 0,C 180,E1 -10800.996,E2 -10800.996} C_VEL
LIN {X 0,Y 404.364,Z 398.096,A -85,B 0,C 180,E1 -10802.989,E2 -10802.989} C_VEL
LIN {X 0,Y 404.38,Z 398.115,A -85,B 0,C 180,E1 -10805.986,E2 -10805.986} C_VEL
LIN {X 0,Y 404.259,Z 398.115,A -85,B 0,C 180,E1 -10809.002,E2 -10809.002} C_VEL
LIN {X 0,Y 404.252,Z 398.129,A -85,B 0,C 180,E1 -10812.042,E2 -10812.042} C_VEL
LIN {X 0,Y 404.16,Z 398.135,A -85,B 0,C 180,E1 -10815.12,E2 -10815.12} C_VEL
LIN {X 0,Y 404.13,Z 398.142,A -85,B 0,C 180,E1 -10818.242,E2 -10818.242} C_VEL
LIN {X 0,Y 404.13,Z 398.143,A -85,B 0,C 180,E1 -10821.42,E2 -10821.42} C_VEL
LIN {X 0,Y 404.138,Z 398.138,A -85,B 0,C 180,E1 -10824.668,E2 -10824.668} C_VEL
LIN {X 0,Y 404.104,Z 398.138,A -85,B 0,C 180,E1 -10828.007,E2 -10828.007} C_VEL
LIN {X 0,Y 404.145,Z 398.14,A -85,B 0,C 180,E1 -10830.285,E2 -10830.285} C_VEL
LIN {X 0,Y 404.14,Z 398.135,A -85,B 0,C 180,E1 -10833.813,E2 -10833.813} C_VEL
LIN {X 0,Y 404.132,Z 398.143,A -85,B 0,C 180,E1 -10836.873,E2 -10836.873} C_VEL
LIN {X 0,Y 404.119,Z 398.117,A -85,B 0,C 180,E1 -10840.075,E2 -10840.075} C_VEL
LIN {X 0,Y 404.142,Z 398.126,A -85,B 0,C 180,E1 -10843.081,E2 -10843.081} C_VEL
LIN {X 0,Y 404.121,Z 398.146,A -85,B 0,C 180,E1 -10845.922,E2 -10845.922} C_VEL
LIN {X 0,Y 404.101,Z 398.117,A -85,B 0,C 180,E1 -10848.632,E2 -10848.632} C_VEL
LIN {X 0,Y 404.135,Z 398.142,A -85,B 0,C 180,E1 -10851.496,E2 -10851.496} C_VEL
LIN {X 0,Y 404.172,Z 398.141,A -85,B 0,C 180,E1 -10854.982,E2 -10854.982} C_VEL
LIN {X 0,Y 404.199,Z 398.275,A -85,B 0,C 180,E1 -10857.052,E2 -10857.052} C_VEL
LIN {X 0,Y 408.784,Z 418.511,A -85,B 0,C 180,E1 -10860.661,E2 -10860.661} C_VEL
LIN {X 0,Y 409.468,Z 422.13,A -85,B 0,C 180,E1 -10861.276,E2 -10861.276} C_VEL
LIN {X 0,Y 408.021,Z 440.937,A -85,B 0,C 180,E1 -10864.219,E2 -10864.219} C_VEL
LIN {X 0,Y 406.697,Z 461.377,A -85,B 0,C 180,E1 -10867.387,E2 -10867.387} C_VEL
LIN {X 0,Y 405.755,Z 477.639,A -85,B 0,C 180,E1 -10869.864,E2 -10869.864} C_VEL
LIN {X 0,Y 406.559,Z 488.401,A -85,B 0,C 180,E1 -10870.423,E2 -10870.423} C_VEL
LIN {X 0,Y 409.842,Z 518.507,A -85,B 0,C 180,E1 -10871.132,E2 -10871.132} C_VEL
LIN {X 0,Y 408.783,Z 607.474,A -85,B 0,C 180,E1 -10872.716,E2 -10872.716} C_VEL
LIN {X 0,Y 408.256,Z 621.148,A -85,B 0,C 180,E1 -10873.176,E2 -10873.176} C_VEL
LIN {X 0,Y 407.718,Z 633.436,A -85,B 0,C 180,E1 -10873.797,E2 -10873.797} C_VEL
LIN {X 0,Y 406.976,Z 645.187,A -85,B 0,C 180,E1 -10874.603,E2 -10874.603} C_VEL
LIN {X 0,Y 406.166,Z 656.852,A -85,B 0,C 180,E1 -10875.636,E2 -10875.636} C_VEL
LIN {X 0,Y 405.518,Z 666.607,A -85,B 0,C 180,E1 -10876.724,E2 -10876.724} C_VEL
LIN {X 0,Y 404.777,Z 675.698,A -85,B 0,C 180,E1 -10877.974,E2 -10877.974} C_VEL
LIN {X 0,Y 404.08,Z 684.529,A -85,B 0,C 180,E1 -10879.477,E2 -10879.477} C_VEL
LIN {X 0,Y 403.615,Z 691.603,A -85,B 0,C 180,E1 -10880.984,E2 -10880.984} C_VEL
LIN {X 0,Y 403.223,Z 697.219,A -85,B 0,C 180,E1 -10882.489,E2 -10882.489} C_VEL
LIN {X 0,Y 403.046,Z 701.617,A -85,B 0,C 180,E1 -10883.994,E2 -10883.994} C_VEL
LIN {X 0,Y 403.041,Z 703.932,A -85,B 0,C 180,E1 -10884.998,E2 -10884.998} C_VEL
LIN {X 0,Y 402.923,Z 705.817,A -85,B 0,C 180,E1 -10885.999,E2 -10885.999} C_VEL
LIN {X 0,Y 402.904,Z 707.239,A -85,B 0,C 180,E1 -10887,E2 -10887} C_VEL
LIN {X 0,Y 402.948,Z 708.242,A -85,B 0,C 180,E1 -10888.001,E2 -10888.001} C_VEL
LIN {X 0,Y 402.905,Z 708.855,A -85,B 0,C 180,E1 -10889,E2 -10889} C_VEL
LIN {X 0,Y 402.904,Z 709.074,A -85,B 0,C 180,E1 -10890,E2 -10890} C_VEL
LIN {X 0,Y 402.931,Z 708.853,A -85,B 0,C 180,E1 -10890.999,E2 -10890.999} C_VEL
LIN {X 0,Y 402.952,Z 708.239,A -85,B 0,C 180,E1 -10891.999,E2 -10891.999} C_VEL
LIN {X 0,Y 402.912,Z 707.234,A -85,B 0,C 180,E1 -10892.999,E2 -10892.999} C_VEL
LIN {X 0,Y 402.933,Z 705.809,A -85,B 0,C 180,E1 -10894.001,E2 -10894.001} C_VEL
LIN {X 0,Y 403.069,Z 702.843,A -85,B 0,C 180,E1 -10895.503,E2 -10895.503} C_VEL
LIN {X 0,Y 403.187,Z 698.812,A -85,B 0,C 180,E1 -10897.008,E2 -10897.008} C_VEL
LIN {X 0,Y 403.552,Z 692.591,A -85,B 0,C 180,E1 -10898.765,E2 -10898.765} C_VEL
LIN {X 0,Y 403.98,Z 685.799,A -85,B 0,C 180,E1 -10900.272,E2 -10900.272} C_VEL
LIN {X 0,Y 404.511,Z 678.843,A -85,B 0,C 180,E1 -10901.525,E2 -10901.525} C_VEL
LIN {X 0,Y 405.172,Z 670.432,A -85,B 0,C 180,E1 -10902.777,E2 -10902.777} C_VEL
LIN {X 0,Y 405.931,Z 660.009,A -85,B 0,C 180,E1 -10904.027,E2 -10904.027} C_VEL
LIN {X 0,Y 406.666,Z 649.672,A -85,B 0,C 180,E1 -10905.024,E2 -10905.024} C_VEL
LIN {X 0,Y 407.382,Z 638.265,A -85,B 0,C 180,E1 -10905.895,E2 -10905.895} C_VEL
LIN {X 0,Y 408.068,Z 626.407,A -85,B 0,C 180,E1 -10906.574,E2 -10906.574} C_VEL
LIN {X 0,Y 408.582,Z 613.588,A -85,B 0,C 180,E1 -10907.099,E2 -10907.099} C_VEL
LIN {X 0,Y 408.881,Z 601.58,A -85,B 0,C 180,E1 -10907.409,E2 -10907.409} C_VEL
LIN {X 0,Y 409.23,Z 582.329,A -85,B 0,C 180,E1 -10907.78,E2 -10907.78} C_VEL
LIN {X 0,Y 410.801,Z 517.361,A -85,B 0,C 180,E1 -10909.288,E2 -10909.288} C_VEL
LIN {X 0,Y 408.606,Z 490.468,A -85,B 0,C 180,E1 -10910.144,E2 -10910.144} C_VEL
LIN {X 0,Y 405.996,Z 472.216,A -85,B 0,C 180,E1 -10910.859,E2 -10910.859} C_VEL
LIN {X 0,Y 407.563,Z 450.031,A -85,B 0,C 180,E1 -10914.447,E2 -10914.447} C_VEL
LIN {X 0,Y 409.492,Z 429.936,A -85,B 0,C 180,E1 -10917.884,E2 -10917.884} C_VEL
LIN {X 0,Y 410.146,Z 423.209,A -85,B 0,C 180,E1 -10919.084,E2 -10919.084} C_VEL
LIN {X 0,Y 408.385,Z 413.823,A -85,B 0,C 180,E1 -10921.083,E2 -10921.083} C_VEL
LIN {X 0,Y 405.586,Z 403.102,A -85,B 0,C 180,E1 -10923.676,E2 -10923.676} C_VEL
LIN {X 0,Y 404.171,Z 398.276,A -85,B 0,C 180,E1 -10925.018,E2 -10925.018} C_VEL
LIN {X 0,Y 404.136,Z 398.146,A -85,B 0,C 180,E1 -10928.504,E2 -10928.504} C_VEL
LIN {X 0,Y 404.105,Z 398.15,A -85,B 0,C 180,E1 -10931.597,E2 -10931.597} C_VEL
LIN {X 0,Y 404.143,Z 398.144,A -85,B 0,C 180,E1 -10934.522,E2 -10934.522} C_VEL
LIN {X 0,Y 404.122,Z 398.145,A -85,B 0,C 180,E1 -10937.294,E2 -10937.294} C_VEL
LIN {X 0,Y 404.133,Z 398.143,A -85,B 0,C 180,E1 -10939.951,E2 -10939.951} C_VEL
LIN {X 0,Y 404.134,Z 398.146,A -85,B 0,C 180,E1 -10943.126,E2 -10943.126} C_VEL
LIN {X 0,Y 404.146,Z 398.144,A -85,B 0,C 180,E1 -10946.188,E2 -10946.188} C_VEL
LIN {X 0,Y 404.146,Z 398.143,A -85,B 0,C 180,E1 -10949.715,E2 -10949.715} C_VEL
LIN {X 0,Y 404.137,Z 398.144,A -85,B 0,C 180,E1 -10953.119,E2 -10953.119} C_VEL
LIN {X 0,Y 404.167,Z 398.142,A -85,B 0,C 180,E1 -10956.425,E2 -10956.425} C_VEL
LIN {X 0,Y 404.208,Z 398.364,A -85,B 0,C 180,E1 -10959.352,E2 -10959.352} C_VEL
LIN {X 0,Y 404.462,Z 399.404,A -85,B 0,C 180,E1 -10959.525,E2 -10959.525} C_VEL
LIN {X 0,Y 410.367,Z 411.247,A -85,B 0,C 180,E1 -10960.38,E2 -10960.38} C_VEL
LIN {X 0,Y 412.752,Z 416.684,A -85,B 0,C 180,E1 -10960.712,E2 -10960.712} C_VEL
LIN {X 0,Y 410.901,Z 480.776,A -85,B 0,C 180,E1 -10962.294,E2 -10962.294} C_VEL
LIN {X 0,Y 410.794,Z 494.286,A -85,B 0,C 180,E1 -10962.739,E2 -10962.739} C_VEL
LIN {X 0,Y 410.527,Z 507.204,A -85,B 0,C 180,E1 -10963.368,E2 -10963.368} C_VEL
LIN {X 0,Y 410.018,Z 519.868,A -85,B 0,C 180,E1 -10964.211,E2 -10964.211} C_VEL
LIN {X 0,Y 409.357,Z 531.405,A -85,B 0,C 180,E1 -10965.204,E2 -10965.204} C_VEL
LIN {X 0,Y 408.65,Z 541.652,A -85,B 0,C 180,E1 -10966.321,E2 -10966.321} C_VEL
LIN {X 0,Y 407.939,Z 550.881,A -85,B 0,C 180,E1 -10967.564,E2 -10967.564} C_VEL
LIN {X 0,Y 407.13,Z 559.772,A -85,B 0,C 180,E1 -10969.054,E2 -10969.054} C_VEL
LIN {X 0,Y 406.478,Z 567.129,A -85,B 0,C 180,E1 -10970.613,E2 -10970.613} C_VEL
LIN {X 0,Y 405.856,Z 572.455,A -85,B 0,C 180,E1 -10972.037,E2 -10972.037} C_VEL
LIN {X 0,Y 405.436,Z 576.757,A -85,B 0,C 180,E1 -10973.531,E2 -10973.531} C_VEL
LIN {X 0,Y 404.963,Z 579.954,A -85,B 0,C 180,E1 -10975.022,E2 -10975.022} C_VEL
LIN {X 0,Y 404.833,Z 581.456,A -85,B 0,C 180,E1 -10976.018,E2 -10976.018} C_VEL
LIN {X 0,Y 404.645,Z 582.555,A -85,B 0,C 180,E1 -10977.013,E2 -10977.013} C_VEL
LIN {X 0,Y 404.514,Z 583.24,A -85,B 0,C 180,E1 -10978.009,E2 -10978.009} C_VEL
LIN {X 0,Y 404.313,Z 583.482,A -85,B 0,C 180,E1 -10979.004,E2 -10979.004} C_VEL
LIN {X 0,Y 404.23,Z 583.291,A -85,B 0,C 180,E1 -10980,E2 -10980} C_VEL
LIN {X 0,Y 404.238,Z 582.685,A -85,B 0,C 180,E1 -10980.996,E2 -10980.996} C_VEL
LIN {X 0,Y 404.163,Z 581.655,A -85,B 0,C 180,E1 -10981.993,E2 -10981.993} C_VEL
LIN {X 0,Y 404.291,Z 580.158,A -85,B 0,C 180,E1 -10982.989,E2 -10982.989} C_VEL
LIN {X 0,Y 404.278,Z 577.125,A -85,B 0,C 180,E1 -10984.487,E2 -10984.487} C_VEL
LIN {X 0,Y 404.531,Z 572.99,A -85,B 0,C 180,E1 -10985.983,E2 -10985.983} C_VEL
LIN {X 0,Y 404.895,Z 567.662,A -85,B 0,C 180,E1 -10987.48,E2 -10987.48} C_VEL
LIN {X 0,Y 405.123,Z 561.003,A -85,B 0,C 180,E1 -10988.982,E2 -10988.982} C_VEL
LIN {X 0,Y 405.538,Z 552.649,A -85,B 0,C 180,E1 -10990.484,E2 -10990.484} C_VEL
LIN {X 0,Y 405.931,Z 544.127,A -85,B 0,C 180,E1 -10991.738,E2 -10991.738} C_VEL
LIN {X 0,Y 406.391,Z 533.714,A -85,B 0,C 180,E1 -10992.992,E2 -10992.992} C_VEL
LIN {X 0,Y 406.949,Z 522.28,A -85,B 0,C 180,E1 -10994.089,E2 -10994.089} C_VEL
LIN {X 0,Y 407.296,Z 510.416,A -85,B 0,C 180,E1 -10995.001,E2 -10995.001} C_VEL
LIN {X 0,Y 407.639,Z 497.446,A -85,B 0,C 180,E1 -10995.756,E2 -10995.756} C_VEL
LIN {X 0,Y 407.897,Z 483.931,A -85,B 0,C 180,E1 -10996.324,E2 -10996.324} C_VEL
LIN {X 0,Y 407.923,Z 469.362,A -85,B 0,C 180,E1 -10996.709,E2 -10996.709} C_VEL
LIN {X 0,Y 408.806,Z 412.532,A -85,B 0,C 180,E1 -10997.929,E2 -10997.929} C_VEL
LIN {X 0,Y 404.415,Z 399.171,A -85,B 0,C 180,E1 -10998.398,E2 -10998.398} C_VEL
